# B&R Automation Studio project MotionTestBenchMaster (part 36)

#### FB_MasterAxis.st
```iecst
FUNCTION_BLOCK FB_MasterAxis
	(* The master position is built from the external struct *)
	IF i_xExternalEncoder OR i_xExternalPositionFormat THEN//V4.A.A.1.7.0
		diMasterPosition	:= i_pstExtEncoderPosition;
	ELSE
		diMasterPosition	:= LREAL_TO_DINT(i_pstMasterPositionStruct.VLab_LRealPosition * 100); //0..36000 * 100 to reach 0..3600000
	END_IF

	IF i_uiNumberOfSteps = 0 THEN
		i_uiNumberOfSteps := 1;
	END_IF

	IF i_udiExternalSignalPeriod = 0 THEN
		i_udiExternalSignalPeriod	:= 3600000;
	END_IF

	(* Master communication fault, Master Encoder not referenced *)
	IF eDigitalSynchroStep > SYNCHRO_INIT THEN
		IF NOT i_xEnable THEN	//V4.A.A.1.6.10
			eDigitalSynchroStep := SYNCHRO_INIT;
		ELSIF NOT i_xCmdEnableCurves AND eDigitalSynchroStep < ERROR THEN
			eDigitalSynchroStep	:= ERROR;
		ELSIF fbWriteParID.Error THEN //Read ParID error
			eDigitalSynchroStep	:= ERROR;
		ELSIF fbCyclicWrite_ExtrEncPos.Error	OR fbCyclicWrite_RefExtrEncPos.Error
			OR fbCyclicRead_ScaledPos.Error		OR fbCyclicRead_ModuloPos.Error 		OR fbCyclicRead_RefModuloPos.Error THEN //Cyclic communication error

			eDigitalSynchroStep	:= ERROR;
		END_IF
	END_IF

	fbRTInfo.enable	:= TRUE;	//V4.A.A.1.6.10
	fbRTInfo();	//V4.A.A.1.6.10

	CASE eDigitalSynchroStep OF
		SYNCHRO_INIT:
			i_pstParameter.i_pdiMasterScaledPos	:= ADR(diMasterScaledPos);
			i_pstParameter.i_plrMasterPosition	:= ADR(lrExternalRefPosition);
			i_pstParameter.i_prMasterVelocity	:= ADR(rExternalRefVelocity);
			i_pstParameter.i_xMachineMaster		:= TRUE;

			i_pstParameter.i_uiMasterParId		:= ACP10PAR_CURVE_VALUE_I4 + 1;

			TON_WaitCurveStabilization.PT		:= T#500ms; // Wait for CURVE FBK stable output
			TON_WaitCurveStabilization.IN		:= FALSE;

			fbPeriodicToContinuePosition.i_xEnable 	:= FALSE;

			(* === Parameters for cyclic data exchange between plc and drive === *)
			fbCyclicRead_ScaledPos.Axis				:= i_pAxisADR;
			fbCyclicRead_ScaledPos.ParID			:= ACP10PAR_CURVE_VALUE_I4 +1;
			fbCyclicRead_ScaledPos.DataAddress		:= ADR(diMasterScaledPos);
			fbCyclicRead_ScaledPos.DataType			:= ncPAR_TYP_DINT;
			fbCyclicRead_ScaledPos.Mode				:= mcEVERY_RECORD;
			fbCyclicRead_ScaledPos.Enable			:= FALSE;

			fbCyclicRead_ModuloPos.Axis				:= i_pAxisADR;
			fbCyclicRead_ModuloPos.ParID			:= ACP10PAR_CURVE_VALUE_REL_I4 +1;
			fbCyclicRead_ModuloPos.DataAddress		:= ADR(diMasterModuloPos);
			fbCyclicRead_ModuloPos.DataType			:= ncPAR_TYP_DINT;
			fbCyclicRead_ModuloPos.Mode				:= mcEVERY_RECORD;
			fbCyclicRead_ModuloPos.Enable			:= FALSE;

			fbCyclicWrite_ExtrEncPos.Axis			:= i_pAxisADR;
			fbCyclicWrite_ExtrEncPos.ParID			:= ACP10PAR_VAR_I4_0;
			fbCyclicWrite_ExtrEncPos.DataAddress	:= ADR(diMasterPosToSpt);
			fbCyclicWrite_ExtrEncPos.DataType		:= ncPAR_TYP_DINT;
			fbCyclicWrite_ExtrEncPos.Mode			:= mcEVERY_RECORD;
			fbCyclicWrite_ExtrEncPos.Enable			:= FALSE;

			(* === Non - Filtered parameter computation for positioning error check === *)
			fbCyclicWrite_RefExtrEncPos.Axis		:= i_pAxisADR;
			fbCyclicWrite_RefExtrEncPos.ParID		:= ACP10PAR_VAR_I4_3;
			fbCyclicWrite_RefExtrEncPos.DataAddress	:= ADR(diRefExtrEncPos);
			fbCyclicWrite_RefExtrEncPos.DataType	:= ncPAR_TYP_DINT;
			fbCyclicWrite_RefExtrEncPos.Mode		:= mcEVERY_RECORD;
			fbCyclicWrite_RefExtrEncPos.Enable		:= FALSE;

			fbCyclicRead_RefModuloPos.Axis			:= i_pAxisADR;
			fbCyclicRead_RefModuloPos.ParID			:= ACP10PAR_CURVE_VALUE_REL_I4 +4;
			fbCyclicRead_RefModuloPos.DataAddress	:= ADR(diRefModuloPos);
			fbCyclicRead_RefModuloPos.DataType		:= ncPAR_TYP_DINT;
//			fbCyclicRead_RefModuloPos.Mode			:= mcEVERY_RECORD;	V 1.1
			fbCyclicRead_RefModuloPos.Enable		:= FALSE;

			IF i_xEnable THEN
				eDigitalSynchroStep		:= CURVES_DISABLE;
			END_IF

		CURVES_DISABLE:
			IF NOT fbWriteParID.Busy THEN
				uiCurveMode					:= 0; //DISABLE
				fbWriteParID.Axis			:= i_pAxisADR;
				fbWriteParID.DataAddress	:= ADR(uiCurveMode);
				fbWriteParID.DataType		:= ncPAR_TYP_UINT;
				fbWriteParID.ParID			:= ACP10PAR_CURVE_MODE + 0;
				fbWriteParID.Execute		:= TRUE;
			END_IF

			IF fbWriteParID.Done AND fbWriteParID.ParID = ACP10PAR_CURVE_MODE + 0 THEN
				fbWriteParID.Execute	:= FALSE;
				eDigitalSynchroStep		:= CURVES_DISABLE_1;
			END_IF

		CURVES_DISABLE_1:
			IF NOT fbWriteParID.Busy THEN
				uiCurveMode					:= 0; //DISABLE
				fbWriteParID.DataAddress	:= ADR(uiCurveMode);
				fbWriteParID.DataType		:= ncPAR_TYP_UINT;
				fbWriteParID.ParID			:= ACP10PAR_CURVE_MODE + 1;
				fbWriteParID.Execute		:= TRUE;
			END_IF

			IF fbWriteParID.Done AND fbWriteParID.ParID = ACP10PAR_CURVE_MODE + 1 THEN
				fbWriteParID.Execute	:= FALSE;
				eDigitalSynchroStep		:= CURVES_DISABLE_2;
			END_IF

		CURVES_DISABLE_2:
			IF NOT fbWriteParID.Busy THEN
				uiCurveMode					:= 0; //DISABLE
				fbWriteParID.DataAddress	:= ADR(uiCurveMode);
				fbWriteParID.DataType		:= ncPAR_TYP_UINT;
				fbWriteParID.ParID			:= ACP10PAR_CURVE_MODE + 3;
				fbWriteParID.Execute		:= TRUE;
			END_IF

			IF fbWriteParID.Done AND fbWriteParID.ParID = ACP10PAR_CURVE_MODE + 3 THEN
				fbWriteParID.Execute	:= FALSE;
				eDigitalSynchroStep		:= CURVES_DISABLE_3;
			END_IF

		CURVES_DISABLE_3:
			IF NOT fbWriteParID.Busy THEN
				uiCurveMode					:= 0; //DISABLE
				fbWriteParID.DataAddress	:= ADR(uiCurveMode);
				fbWriteParID.DataType		:= ncPAR_TYP_UINT;
				fbWriteParID.ParID			:= ACP10PAR_CURVE_MODE + 4;
				fbWriteParID.Execute		:= TRUE;
			END_IF

			IF fbWriteParID.Done AND fbWriteParID.ParID = ACP10PAR_CURVE_MODE + 4 THEN
				TON_WaitCurveStabilization.IN	:= FALSE;
				fbWriteParID.Execute			:= FALSE;
				eDigitalSynchroStep				:= ZERO_OFFSET;
			END_IF

		(* In order to be sure that the OFFSET is zero at the startup the value is force *)
		ZERO_OFFSET:
			IF NOT fbWriteParID.Busy THEN
				q_diOffsetModuloPos			:= 0;
				fbWriteParID.DataAddress	:= ADR(q_diOffsetModuloPos);
				fbWriteParID.DataType		:= ncPAR_TYP_DINT;
				fbWriteParID.ParID			:= ACP10PAR_VAR_I4_1 +0;
				fbWriteParID.Execute		:= TRUE;
			END_IF

			IF fbWriteParID.Done AND fbWriteParID.ParID = ACP10PAR_VAR_I4_1 + 0 THEN
				fbWriteParID.Execute 	:= FALSE;
				q_xPositionRestored 	:= TRUE;
				eDigitalSynchroStep 	:= WRITE_MA_PERIOD;
			END_IF

		WRITE_MA_PERIOD:
			IF NOT fbWriteParID.Busy THEN
				diMasterPeriod				:= i_udiExternalSignalPeriod;
				fbWriteParID.Axis			:= i_pAxisADR;
				fbWriteParID.DataAddress	:= ADR(diMasterPeriod);
				fbWriteParID.DataType		:= ncPAR_TYP_DINT;
				fbWriteParID.ParID			:= ACP10PAR_CURVE_X_FACTOR + 0;
				fbWriteParID.Execute		:= TRUE;
			END_IF

			IF fbWriteParID.Done AND fbWriteParID.ParID = ACP10PAR_CURVE_X_FACTOR + 0 THEN
				fbWriteParID.Execute	:= FALSE;
				eDigitalSynchroStep		:= WRITE_MA_PERIOD_1;
			END_IF

		WRITE_MA_PERIOD_1:
			IF NOT fbWriteParID.Busy THEN
				diMasterPeriod				:= i_udiExternalSignalPeriod;
				fbWriteParID.Axis			:= i_pAxisADR;
				fbWriteParID.DataAddress	:= ADR(diMasterPeriod);
				fbWriteParID.DataType		:= ncPAR_TYP_DINT;
				fbWriteParID.ParID			:= ACP10PAR_CURVE_X_FACTOR + 3;
				fbWriteParID.Execute		:= TRUE;
			END_IF

			IF fbWriteParID.Done AND fbWriteParID.ParID = ACP10PAR_CURVE_X_FACTOR + 3 THEN
				fbWriteParID.Execute	:= FALSE;
				eDigitalSynchroStep		:= WRITE_SL_PERIOD;
			END_IF

		WRITE_SL_PERIOD:
			IF NOT fbWriteParID.Busy THEN
				diSlavePeriod				:= i_uiNumberOfSteps * 360 * c_uiAxisFactor;
				fbWriteParID.Axis			:= i_pAxisADR;
				fbWriteParID.DataAddress	:= ADR(diSlavePeriod);
				fbWriteParID.DataType		:= ncPAR_TYP_DINT;
				fbWriteParID.ParID			:= ACP10PAR_CURVE_Y_FACTOR + 0;
				fbWriteParID.Execute		:= TRUE;
			END_IF

			IF fbWriteParID.Done AND fbWriteParID.ParID = ACP10PAR_CURVE_Y_FACTOR + 0 THEN
				fbWriteParID.Execute	:= FALSE;
				eDigitalSynchroStep		:= WRITE_SL_PERIOD_1;
			END_IF

		WRITE_SL_PERIOD_1:
			IF NOT fbWriteParID.Busy THEN
				diSlavePeriod				:= i_uiNumberOfSteps * 360 * c_uiAxisFactor;
				fbWriteParID.Axis			:= i_pAxisADR;
				fbWriteParID.DataAddress	:= ADR(diSlavePeriod);
				fbWriteParID.DataType		:= ncPAR_TYP_DINT;
				fbWriteParID.ParID			:= ACP10PAR_CURVE_Y_FACTOR + 3;
				fbWriteParID.Execute		:= TRUE;
			END_IF

			IF fbWriteParID.Done AND fbWriteParID.ParID = ACP10PAR_CURVE_Y_FACTOR + 3 THEN
				fbWriteParID.Execute	:= FALSE;
				eDigitalSynchroStep		:= INIT_FILTERS;
			END_IF

		INIT_FILTERS:
			lrFilterTime 	:= UINT_TO_LREAL(i_uiFilteringCoefficient) * c_rTf_min; (* s *)
			lrExtrTime 		:= (UDINT_TO_LREAL(fbRTInfo.cycle_time) / 1E6) * UINT_TO_LREAL(i_uiNumberOfEplCycles) + c_timCompensationIPL; (* s *)	//V4.A.A.1.6.10

			(* Periodic to continue position enable *)
			fbPeriodicToContinuePosition.i_xEnable 	:= TRUE;

			(* Reference filter enable *)
			(* The enable is done only in case of i_uiFilteringCoefficient > 0 *)

			fbEXTR_RefFilter.Enable		:= lrFilterTime > 0;

			(* Extrapolation filter enable *)
			fbPT1_EncFilter.Enable 		:= fbEXTR_RefFilter.Enable;

			IF i_udiExternalSignalPeriod > 0 THEN
				diInitialOffset	:= diMasterPosition - (diMasterPosition MOD UDINT_TO_DINT(i_udiExternalSignalPeriod));
			END_IF

			IF fbEXTR_RefFilter.Enable AND fbPT1_EncFilter.Enable THEN
				IF fbPT1_EncFilter.Valid THEN
					fbEXTR_EncFilter.Enable	:= TRUE;
					IF fbEXTR_EncFilter.Valid AND fbEXTR_RefFilter.Valid THEN
						TON_WaitCurveStabilization.IN	:= FALSE;
						eDigitalSynchroStep 			:= DISABLE_IPL;
					END_IF
				END_IF
			ELSE
				TON_WaitCurveStabilization.IN	:= FALSE;
				eDigitalSynchroStep 			:= DISABLE_IPL;
			END_IF

		DISABLE_IPL:
			IF NOT fbWriteParID.Busy THEN
				uiIPLMode					:= 0;
				fbWriteParID.Axis			:= i_pAxisADR;
				fbWriteParID.DataAddress	:= ADR(uiIPLMode);
				fbWriteParID.DataType		:= ncPAR_TYP_UINT;
				fbWriteParID.ParID			:= ACP10PAR_IPL_MODE + 0;
				fbWriteParID.Execute		:= TRUE;
			END_IF

			TON_WaitCurveStabilization.IN	:= fbWriteParID.Done;
			TON_WaitCurveStabilization.PT	:= T#0.5S;

			IF TON_WaitCurveStabilization.Q AND fbWriteParID.ParID = ACP10PAR_IPL_MODE + 0 THEN
				fbWriteParID.Execute	:= FALSE;
				eDigitalSynchroStep		:= INIT_CYCLIC_READ_WRITE;
			END_IF

		INIT_CYCLIC_READ_WRITE:
			fbCyclicWrite_ExtrEncPos.Enable		:= TRUE;
			fbCyclicWrite_RefExtrEncPos.Enable	:= TRUE;

			fbCyclicRead_ScaledPos.Enable		:= TRUE;
			fbCyclicRead_ModuloPos.Enable 		:= TRUE;
			fbCyclicRead_RefModuloPos.Enable	:= TRUE;

			q_xCyclicComValid	:= fbCyclicWrite_ExtrEncPos.Valid AND fbCyclicWrite_RefExtrEncPos.Valid AND fbCyclicRead_ScaledPos.Valid AND
									fbCyclicRead_ModuloPos.Valid AND fbCyclicRead_RefModuloPos.Valid;

			IF fbCyclicWrite_ExtrEncPos.Error OR fbCyclicWrite_RefExtrEncPos.Error OR fbCyclicRead_ScaledPos.Error OR fbCyclicRead_ModuloPos.Error OR fbCyclicRead_RefModuloPos.Error THEN
				q_xCyclicComValid 	:= FALSE;
				eDigitalSynchroStep := ERROR;
			ELSIF q_xCyclicComValid THEN
				TON_WaitCurveStabilization.IN	:= FALSE;
				eDigitalSynchroStep 			:= WRITE_IPL_CYCLIE_TIME;
			END_IF

		WRITE_IPL_CYCLIE_TIME:
			IF NOT fbWriteParID.Busy THEN

				IF i_xExternalEncoder THEN
					udiCycleTime				:= fbRTInfo.cycle_time * 10;	//V4.A.A.1.6.10
				ELSIF i_xExternalPositionFormat THEN//V4.A.A.1.7.0
					udiCycleTime				:= fbRTInfo.cycle_time * 2;//V4.A.A.1.7.0
				ELSE
					udiCycleTime				:= fbRTInfo.cycle_time;	//V4.A.A.1.6.10
				END_IF

				fbWriteParID.Axis			:= i_pAxisADR;
				fbWriteParID.DataAddress	:= ADR(udiCycleTime);
				fbWriteParID.DataType		:= ncPAR_TYP_UDINT;
				fbWriteParID.ParID			:= ACP10PAR_IPL_CYCLE_TIME + 0;
				fbWriteParID.Execute		:= TRUE;
			END_IF

			IF fbWriteParID.Done AND fbWriteParID.ParID = ACP10PAR_IPL_CYCLE_TIME + 0 THEN
				fbWriteParID.Execute	:= FALSE;
				eDigitalSynchroStep		:= ENABLE_IPL;
			END_IF

		ENABLE_IPL:
			IF NOT fbWriteParID.Busy THEN
				uiIPLMode					:= 1;
				fbWriteParID.Axis			:= i_pAxisADR;
				fbWriteParID.DataAddress	:= ADR(uiIPLMode);
				fbWriteParID.DataType		:= ncPAR_TYP_UINT;
				fbWriteParID.ParID			:= ACP10PAR_IPL_MODE + 0;
				fbWriteParID.Execute		:= TRUE;
			END_IF

			TON_WaitCurveStabilization.IN	:= fbWriteParID.Done;
			TON_WaitCurveStabilization.PT	:= T#0.5S;

			IF TON_WaitCurveStabilization.Q AND fbWriteParID.ParID = ACP10PAR_IPL_MODE + 0 THEN
				fbWriteParID.Execute	:= FALSE;
				eDigitalSynchroStep		:= CURVES_ENABLE;
			END_IF

		CURVES_ENABLE:
			IF NOT fbWriteParID.Busy THEN
				uiCurveMode					:= 2;
				fbWriteParID.Axis			:= i_pAxisADR;
				fbWriteParID.DataAddress	:= ADR(uiCurveMode);
				fbWriteParID.DataType		:= ncPAR_TYP_UINT;
				fbWriteParID.ParID			:= ACP10PAR_CURVE_MODE + 0;
				fbWriteParID.Execute		:= TRUE;
			END_IF

			IF fbWriteParID.Done AND fbWriteParID.ParID = ACP10PAR_CURVE_MODE + 0 THEN
				fbWriteParID.Execute	:= FALSE;
				eDigitalSynchroStep		:= CURVES_ENABLE_1;
			END_IF

		CURVES_ENABLE_1:
			IF NOT fbWriteParID.Busy THEN
				uiCurveMode					:= 2;
				fbWriteParID.DataAddress	:= ADR(uiCurveMode);
				fbWriteParID.DataType		:= ncPAR_TYP_UINT;
				fbWriteParID.ParID			:= ACP10PAR_CURVE_MODE + 1;
				fbWriteParID.Execute		:= TRUE;
			END_IF

			IF fbWriteParID.Done AND fbWriteParID.ParID = ACP10PAR_CURVE_MODE + 1 THEN
				fbWriteParID.Execute	:= FALSE;
				eDigitalSynchroStep		:= CURVES_ENABLE_2;
			END_IF

		CURVES_ENABLE_2:
			IF NOT fbWriteParID.Busy THEN
				uiCurveMode					:= 2;
				fbWriteParID.DataAddress	:= ADR(uiCurveMode);
				fbWriteParID.DataType		:= ncPAR_TYP_UINT;
				fbWriteParID.ParID			:= ACP10PAR_CURVE_MODE + 3;
				fbWriteParID.Execute		:= TRUE;
			END_IF

			IF fbWriteParID.Done AND fbWriteParID.ParID = ACP10PAR_CURVE_MODE + 3 THEN
				fbWriteParID.Execute	:= FALSE;
				eDigitalSynchroStep		:= CURVES_ENABLE_3;
			END_IF

		CURVES_ENABLE_3:
			IF NOT fbWriteParID.Busy THEN
				uiCurveMode					:= 2;
				fbWriteParID.DataAddress	:= ADR(uiCurveMode);
				fbWriteParID.DataType		:= ncPAR_TYP_UINT;
				fbWriteParID.ParID			:= ACP10PAR_CURVE_MODE + 4;
				fbWriteParID.Execute		:= TRUE;
			END_IF

			IF fbWriteParID.Done AND fbWriteParID.ParID = ACP10PAR_CURVE_MODE + 4 THEN
				fbWriteParID.Execute			:= FALSE;
				TON_WaitCurveStabilization.IN	:= FALSE;
				eDigitalSynchroStep				:= WAIT_CURVES_STABILIZATION;
			END_IF

		WAIT_CURVES_STABILIZATION:
			IF diOldScaledPos = diMasterScaledPos AND diOldModuloPos = diMasterModuloPos THEN
				TON_WaitCurveStabilization.IN	:= TRUE;
				IF TON_WaitCurveStabilization.Q THEN
					TON_WaitCurveStabilization.IN	:= FALSE;
					q_xPositionValid 				:= TRUE;
					eDigitalSynchroStep				:= RESTORE_CALIBRATION_OFFSET;
				END_IF
			ELSE
				TON_WaitCurveStabilization.IN := FALSE;
				diOldScaledPos := diMasterScaledPos;
				diOldModuloPos := diMasterModuloPos;
			END_IF

		RESTORE_CALIBRATION_OFFSET:
			IF NOT fbWriteParID.Busy THEN
				q_diOffsetModuloPos			:= i_pstAbsEncPerm.diAbsEncOffset;
				fbWriteParID.DataAddress	:= ADR(q_diOffsetModuloPos);
				fbWriteParID.DataType		:= ncPAR_TYP_DINT;
				fbWriteParID.ParID			:= ACP10PAR_VAR_I4_1 +0;
				fbWriteParID.Execute		:= TRUE;
			END_IF

			IF fbWriteParID.Done AND fbWriteParID.ParID = ACP10PAR_VAR_I4_1 + 0 THEN
				fbWriteParID.Execute := FALSE;

				q_xPositionRestored := TRUE;
				eDigitalSynchroStep := ABS_ENC_READY;
			END_IF

		ABS_ENC_READY:
			q_xCyclicComValid	:= fbCyclicWrite_ExtrEncPos.Valid AND fbCyclicWrite_RefExtrEncPos.Valid AND fbCyclicRead_ScaledPos.Valid AND
									fbCyclicRead_ModuloPos.Valid AND fbCyclicRead_RefModuloPos.Valid;

			IF NOT q_xCyclicComValid OR NOT i_xCmdEnableCurves THEN
				eDigitalSynchroStep		:= ERROR;
			ELSIF i_pstStatus.q_stMainAxisStatus.q_xSynchroWithOffset AND i_pstCmd.i_xPhaseCompensation THEN //V4.A.A.1.6.10
				eDigitalSynchroStep		:= OFFSET_RESET;
			ELSIF i_xCmdHoming THEN
				eDigitalSynchroStep		:= CALIBRATION;
			END_IF

		OFFSET_RESET:
			q_diOffsetModuloPos	:= REAL_TO_DINT(i_pstAxisHome.rPhaseOffsetValue * c_uiAxisFactor) + i_pstAbsEncPerm.diAbsEncOffset;

			i_pstAxisHome.rPhaseOffsetValue		:= 0;
			i_pstAbsEncPerm.diAbsEncOffset		:= q_diOffsetModuloPos;
			i_pstAbsEncPerm.xCalibrationDone	:= FALSE;
			eDigitalSynchroStep					:= WRITE_NEW_CALIBRATION_VALUE;

		CALIBRATION:
			q_diOffsetModuloPos := LREAL_TO_DINT(i_pstStatus.q_stMainAxisStatus.q_lrPosition * c_uiAxisFactor) - diRefModuloPos;

			IF q_diOffsetModuloPos < 0 THEN
				q_diOffsetModuloPos := q_diOffsetModuloPos + 36000;
			END_IF

			i_pstAbsEncPerm.diAbsEncOffset		:= q_diOffsetModuloPos;
			i_pstAbsEncPerm.xCalibrationDone	:= FALSE;

			eDigitalSynchroStep 	:= WRITE_NEW_CALIBRATION_VALUE;

		WRITE_NEW_CALIBRATION_VALUE:
			IF NOT fbWriteParID.Busy THEN
				fbWriteParID.Axis			:= i_pAxisADR;
				fbWriteParID.DataAddress	:= ADR(q_diOffsetModuloPos);
				fbWriteParID.DataType		:= ncPAR_TYP_DINT;
				fbWriteParID.ParID			:= ACP10PAR_VAR_I4_1;
				fbWriteParID.Execute		:= TRUE;
			END_IF

			IF fbWriteParID.Done AND fbWriteParID.ParID = ACP10PAR_VAR_I4_1 AND NOT i_pstCmd.i_xPhaseCompensation AND NOT i_xCmdHoming THEN
				fbWriteParID.Execute 				:= FALSE;
				i_pstAbsEncPerm.xCalibrationDone	:= TRUE;
				q_xPositionRestored					:= TRUE;
				eDigitalSynchroStep					:= WAIT_CURVES_STABILIZATION;
			END_IF

		(*****************************************)
		ERROR:
			q_xPositionRestored						:= FALSE;
			q_xCyclicComValid						:= FALSE;
			q_xPositionValid  						:= FALSE;

			TON_WaitCurveStabilization.IN 			:= FALSE;
			fbPeriodicToContinuePosition.i_xEnable 	:= FALSE;

			IF i_pstCmd.i_xErrorReset THEN
				fbCyclicWrite_ExtrEncPos.Enable		:= FALSE;
				fbCyclicWrite_RefExtrEncPos.Enable	:= FALSE;

				fbCyclicRead_ScaledPos.Enable		:= FALSE;
				fbCyclicRead_ModuloPos.Enable 		:= FALSE;
				fbCyclicRead_RefModuloPos.Enable	:= FALSE;

				fbPT1_EncFilter.Enable 	:= FALSE;
				fbEXTR_EncFilter.Enable	:= FALSE;
				fbEXTR_RefFilter.Enable	:= FALSE;
				IF fbWriteParID.Error THEN
					fbWriteParID.Execute := FALSE;
				END_IF
			END_IF

			IF NOT fbCyclicWrite_ExtrEncPos.Error AND NOT fbCyclicWrite_RefExtrEncPos.Error AND NOT fbCyclicRead_ScaledPos.Error AND
				NOT fbCyclicRead_ModuloPos.Error AND NOT fbCyclicRead_RefModuloPos.Error AND NOT fbWriteParID.Error THEN

				eDigitalSynchroStep := ERROR_1;
			END_IF

		ERROR_1: (* Wait Master data are OK *)
			IF i_xCmdEnableCurves THEN
				eDigitalSynchroStep := CURVES_DISABLE;
			END_IF
	END_CASE

	(* Timer for curve stabilization *)
	TON_WaitCurveStabilization();

	fbWriteParID();

	fbCyclicRead_ScaledPos();
	fbCyclicRead_ModuloPos();
	fbCyclicRead_RefModuloPos();
	fbCyclicWrite_ExtrEncPos();
	fbCyclicWrite_RefExtrEncPos();

	(* Periodic TO Continue DINT position *)
	IF NOT i_xExternalEncoder THEN
		fbPeriodicToContinuePosition.i_diInPosition	:= diMasterPosition;
		fbPeriodicToContinuePosition.i_udiPeriod	:= i_udiExternalSignalPeriod;
		fbPeriodicToContinuePosition();
	END_IF

	IF fbPT1_EncFilter.Enable THEN
		IF NOT i_xExternalEncoder THEN (* External Value filtering *)
			fbPT1_EncFilter.T1	:= lrFilterTime;
			fbPT1_EncFilter.U	:= fbPeriodicToContinuePosition.q_diPosition;
		ELSE (* External Value filtering *)
			fbPT1_EncFilter.T1	:= lrFilterTime;
			fbPT1_EncFilter.U	:= (diMasterPosition - diInitialOffset);
		END_IF

		fbPT1_EncFilter();

		(* External value extrapolation *)
		fbEXTR_EncFilter.T_ext	:= lrExtrTime + lrFilterTime;
		fbEXTR_EncFilter.U		:= fbPT1_EncFilter.X;
		fbEXTR_EncFilter();

		(* External Value filtering *)
		IF NOT i_xExternalEncoder THEN
			diMasterPosToSpt	 	:= fbEXTR_EncFilter.X;
		ELSE
			uiMasterPositionSampling := uiMasterPositionSampling + 1;	//v1.2
			IF uiMasterPositionSampling >= 10 THEN				//v1.2
				diMasterPosToSpt	 	:= fbEXTR_EncFilter.X;
				uiMasterPositionSampling	:= 0;			//v1.2
			END_IF
		END_IF

		(* Non-filtered position extrapolation *)
		IF NOT i_xExternalEncoder THEN (* External Value filtering *)
			fbEXTR_RefFilter.T_ext	:= lrExtrTime;
			fbEXTR_RefFilter.U	:= fbPeriodicToContinuePosition.q_diPosition;
		ELSE (* External Value filtering *)
			fbEXTR_RefFilter.T_ext	:= lrExtrTime;
			fbEXTR_RefFilter.U	:= (diMasterPosition - diInitialOffset);
		END_IF
		fbEXTR_RefFilter();

		diRefExtrEncPos			:= fbEXTR_RefFilter.X;

		(* Extrapolation error computing *)
		IF EDGEPOS(q_xPositionValid) THEN
			diRefModuloOffset := diMasterModuloPos - diRefModuloPos;
		END_IF

		q_diRefPosError := diMasterModuloPos - diRefModuloPos - diRefModuloOffset;

		IF ABS(q_diRefPosError + 360 * c_uiAxisFactor) < ABS(q_diRefPosError) THEN
			q_diRefPosError := q_diRefPosError + 360 * c_uiAxisFactor;
		ELSIF ABS(q_diRefPosError - 360 * c_uiAxisFactor) < ABS(q_diRefPosError) THEN
			q_diRefPosError := q_diRefPosError - 360 * c_uiAxisFactor;
		END_IF
	ELSIF NOT i_xExternalEncoder THEN
		diMasterPosToSpt	:= fbPeriodicToContinuePosition.q_diPosition;
		diRefExtrEncPos		:= fbPeriodicToContinuePosition.q_diPosition;
	ELSE
		uiMasterPositionSampling := uiMasterPositionSampling + 1;	//v1.2
		IF uiMasterPositionSampling >= 10 THEN				//v1.2
			diMasterPosToSpt	 	:= diMasterPosition;
			uiMasterPositionSampling	:= 0;			//v1.2
		END_IF

		diRefExtrEncPos		:= diMasterPosition;
	END_IF

	(* External reference position and velocity *)
	lrExternalRefPosition  := UDINT_TO_LREAL(diMasterModuloPos) / c_uiAxisFactor;

	fbVelocity.i_diPosition	:= diMasterScaledPos;
	fbVelocity();
	rExternalRefVelocity	:= fbVelocity.q_rVelocity / c_uiAxisFactor;
END_FUNCTION_BLOCK
```

#### FB_Step2PeriodicPosition.st
```iecst
(* From a step signal a periodic signal is created *)
FUNCTION_BLOCK FB_PeriodicPosition
	IF NOT i_xEnable OR i_rPeriod <=0 THEN
		usiStep				:= 0;
		q_xPositionValid	:= FALSE;
	ELSE
		CASE usiStep OF
			0:
				q_xPositionValid	:= FALSE;
				q_rPeriodicPosition	:= 0;
				rPosition			:= 0;

				IF i_xEnable THEN
					usiStep	:= 10;
				END_IF

			10:
				IF EDGEPOS(i_xResetPostion) THEN
					q_xPositionValid	:= TRUE;
					rPosition			:= i_rAxisPosition;
					q_rPeriodicPosition	:= i_rAxisPosition;
					usiStep				:= 20;
				END_IF

			20:
				rDeltaPos	:= i_rAxisPosition - rPosition;
				// If the difference between the old axis and the current axis position
				// If greater than 180° it means that we overlapped the period
				IF ABS(rDeltaPos) > 180 THEN
					IF rDeltaPos > 0 THEN
						rDeltaPos	:= rDeltaPos - 360;
					ELSE
						rDeltaPos	:= rDeltaPos + 360;
					END_IF
				END_IF

				q_rPeriodicPosition	:= FC_RealReminder(q_rPeriodicPosition + rDeltaPos, i_rPeriod, 0);
				rPosition			:= i_rAxisPosition;

				IF i_xResetPostion	THEN
					usiStep	:= 0;
				END_IF
		END_CASE
	END_IF
END_FUNCTION_BLOCK
```

#### FB_CamGenerator.st
```iecst
(* Cam Generator Function Block *)
FUNCTION_BLOCK FB_CamGenerator
	IF i_xEnable AND i_usiNumberOfPulse > 0 THEN
		IF i_usiNumberOfPulse = 1 AND i_rOnPosition <> i_rOffPosition THEN
			rAdvPosition		:= i_rAdvanceTime * i_prAxisVelocity / 1000.0;
			q_xAdvError			:= (ABS(rAdvPosition) >= 360);

			i_pxPointerStepAdv	:= ((i_rOnPosition - rAdvPosition) < 0);

			rOnPositionA		:= FC_RealReminder(i_rOnPosition - rAdvPosition,	360.0, 0);
			rOffPositionA		:= FC_RealReminder(i_rOffPosition - rAdvPosition,	360.0, 0);

			(* CAM A GENERATION *)
			IF(rOnPositionA < rOffPositionA) THEN
				xCamValueA	:= (i_plrAxisPosition >= rOnPositionA) AND (i_plrAxisPosition < rOffPositionA);
			ELSE
				xCamValueA	:= i_plrAxisPosition >= rOnPositionA OR i_plrAxisPosition < rOffPositionA;
			END_IF

			IF xCamValueA <> xOldCamValueA THEN
				rTempReal	:= SEL(xCamValueA, rOffPositionA, rOnPositionA);
				rTempReal	:= rTempReal - LREAL_TO_REAL(i_plrAxisPosition);
				IF ABS(rTempReal) > 0.5 AND ABS(rTempReal) < 359.5 THEN
					xOldCamValueA := xCamValueA;
				END_IF
			END_IF

			(* CAM B GENERATION *)
			IF i_rOnPositionB <> 0 AND i_rOffPositionB <> 0 THEN
				rOnPositionB		:= FC_RealReminder(i_rOnPositionB - rAdvPosition,	360.0, 0);
				rOffPositionB		:= FC_RealReminder(i_rOffPositionB - rAdvPosition,	360.0, 0);
				IF(rOnPositionB < rOffPositionB) THEN
					xCamValueB	:= (i_plrAxisPosition >= rOnPositionB) AND (i_plrAxisPosition < rOffPositionB);
				ELSE
					xCamValueB	:= i_plrAxisPosition >= rOnPositionB OR i_plrAxisPosition < rOffPositionB;
				END_IF

				IF xCamValueB <> xOldCamValueB THEN
					rTempReal	:= SEL(xCamValueB, rOffPositionB, rOnPositionB);
					rTempReal	:= rTempReal - LREAL_TO_REAL(i_plrAxisPosition);
					IF ABS(rTempReal) > 0.5 AND ABS(rTempReal) < 359.5 THEN
						xOldCamValueB	:=	xCamValueB;
					END_IF
				END_IF

				(* Debounce *)
				CASE usiStep OF
					0:(* INIT *)
						usiStep := 100;

					100:(* WAIT FOR CAM A RAISING EDGE *)
						IF xCamValueA THEN
							i_pxPointerOutput := TRUE;
							usiStep := 110;
						END_IF

					110:(* WAIT FOR CAM B FALLING EDGE *)
						IF NOT xCamValueB THEN
							usiStep := 120;
						END_IF

					120:(*  WAIT FOR CAM A FALLING EDGE *)
						IF NOT xCamValueA THEN
							i_pxPointerOutput := FALSE;
							usiStep := 130;
						END_IF

					130:(* WAIT FOR CAM B RAISING EDGE *)
						IF xCamValueB THEN
							usiStep := 100;
						END_IF

					ELSE
						usiStep := 200;
				END_CASE
			ELSE
				(* Simple cam A generator *)
				i_pxPointerOutput	:= xOldCamValueA;
			END_IF
		ELSIF i_usiNumberOfPulse <= 10 THEN
			i_pxPointerStepAdv	:= FALSE;
			i_pxPointerOutput	:= FC_RealReminder(LREAL_TO_REAL(i_plrAxisPosition), 360.0 / i_usiNumberOfPulse, 0) >= 180.0 / i_usiNumberOfPulse;
		END_IF
	ELSE
		i_pxPointerOutput	:= FALSE;
		q_xAdvError			:= FALSE;
	END_IF
END_FUNCTION_BLOCK

(* Cam Generator Function Block *)
FUNCTION_BLOCK FB_CamGenerator_v2
	IF i_xEnable AND i_usiNumberOfPulse > 0 THEN
		IF i_usiNumberOfPulse = 1 AND i_rOnPosition <> i_rOffPosition THEN
			rPosition			:= DINT_TO_REAL(i_pdiAxisPosition MOD 36000) / 100.0;
			rAdvPosition		:= i_rAdvanceTime * i_prAxisVelocity / 100000.0; //v1.4
			q_xAdvError			:= (ABS(rAdvPosition) >= 360);

			i_pxPointerStepAdv	:= ((i_rOnPosition - rAdvPosition) < 0);

			rOnPosition		:= FC_RealReminder(i_rOnPosition - rAdvPosition,	360.0, 0);
			rOffPosition	:= FC_RealReminder(i_rOffPosition - rAdvPosition,	360.0, 0);

			(* CAM GENERATION *)
			IF(rOnPosition < rOffPosition) THEN
				xCamValue	:= (rPosition >= rOnPosition) AND (rPosition < rOffPosition);
			ELSE
				xCamValue	:= rPosition >= rOnPosition OR rPosition < rOffPosition;
			END_IF

			IF xCamValue <> xOldCamValue THEN
				rTempReal	:= SEL(xCamValue, rOffPosition, rOnPosition);
				rTempReal	:= rTempReal - rPosition;
				IF ABS(rTempReal) > 0.5 AND ABS(rTempReal) < 359.5 THEN
					xOldCamValue := xCamValue;
				END_IF
			END_IF

			i_pxPointerOutput	:= xOldCamValue;
		ELSIF i_usiNumberOfPulse <= 10 THEN
			i_pxPointerStepAdv	:= FALSE;
			rPosition			:= DINT_TO_REAL(i_pdiAxisPosition MOD 36000) / 100.0;
			i_pxPointerOutput	:= FC_RealReminder(rPosition, 360.0 / i_usiNumberOfPulse, 0) >= 180.0 / i_usiNumberOfPulse;
		END_IF
	ELSE
		i_pxPointerOutput	:= FALSE;
		q_xAdvError			:= FALSE;
	END_IF
END_FUNCTION_BLOCK
```

#### FB_ExceptionAlarmX.st
```iecst
(* Fb for mananging alarms *)
FUNCTION_BLOCK FB_ExceptionAlarmX
	IF i_pxInitCoreDone THEN
		IF i_xConditions AND NOT xAlarmActive THEN
			xAlarmActive := TRUE;
			MpAlarmXSet(MpLink := i_pstMpAlarmXLink, Name := i_psAlarmName);
		ELSIF NOT i_xConditions AND xAlarmActive THEN
			IF i_pxAcknowledge OR i_xAutoAck THEN
				xAlarmActive := FALSE;
				MpAlarmXReset(MpLink := i_pstMpAlarmXLink, Name := i_psAlarmName);
			END_IF
		END_IF
		q_xAlarmActive := xAlarmActive;
	END_IF
END_FUNCTION_BLOCK
```

#### FB_Position2Velocity.st
```iecst
FUNCTION_BLOCK FB_Position2Velocity
	fbRTInfo(enable := TRUE);
	adiBuffer[uiCount]	:= i_diPosition;
	IF uiCount > 0 THEN
		arBufferVel[uiCount] := DINT_TO_REAL((i_diPosition - adiBuffer[uiCount - 1])) / (DINT_TO_REAL(fbRTInfo.cycle_time) * 1E-6);
	ELSE
		arBufferVel[uiCount] := DINT_TO_REAL((i_diPosition - adiBuffer[c_usiNSample - 1])) / (DINT_TO_REAL(fbRTInfo.cycle_time) * 1E-6);
	END_IF

	uiCount 	:= (uiCount + 1) MOD c_usiNSample;
	rInternal	:= 0;

	FOR i := 0 TO c_usiNSample - 1 DO
		rInternal	:= rInternal + arBufferVel[i];
	END_FOR

	q_rVelocity := rInternal / c_usiNSample;
END_FUNCTION_BLOCK
```

#### FB_Periodic2ContinuePosition.st
```iecst
FUNCTION_BLOCK FB_Periodic2ContinuePosition
	IF NOT i_xEnable THEN
		xActive 		:= FALSE;
		diOldInPosition := 0;
		q_diPosition	:= 0;
		RETURN;
	ELSIF NOT xActive THEN
		xActive 		:= TRUE;
		q_diPosition	:= i_diInPosition;
		diOldInPosition := i_diInPosition;
	ELSE
		(* Continue DINT position calculation *)
		IF ABS(i_diInPosition - diOldInPosition) < UDINT_TO_DINT(i_udiPeriod / 2) THEN
			q_diPosition		:= q_diPosition + (i_diInPosition - diOldInPosition);
		ELSIF i_diInPosition < diOldInPosition THEN
			q_diPosition		:= q_diPosition + i_udiPeriod + (i_diInPosition - diOldInPosition);
		ELSE
			q_diPosition		:= q_diPosition - i_udiPeriod + (i_diInPosition - diOldInPosition);
		END_IF
		diOldInPosition 	:= i_diInPosition;
	END_IF
END_FUNCTION_BLOCK
```

#### FB_EncEmul.st
```iecst
(*********************************************************************************
 * Copyright:
 * Author:    		EncoderEmulationManagement
 * Created:  		July 4, 2016/2:37 PM
 * HELP REFERENCE:  ncsoftware/acp10_drivefunctions/acp10_drivefunctions-63-15.html
 *********************************************************************************)

(* Encoder Emulation on 8BAC130.001-1 plug-in module*)
FUNCTION_BLOCK FB_EncEmul
	IF i_pstEncEmulAxis.nc_obj_inf.node_nr > 0 AND i_pstEncEmulAxis.network.phase  <> 90 AND uiStep > 0 THEN
		uiStep := 950;
	ELSIF fbAxisError.Error	THEN
		uiStep := 960;
	ELSIF fbAxisError.Enable AND (fbAxisError.FunctionBlockErrorCount > 0 OR fbAxisError.AxisErrorCount > 0 ) THEN
		uiStep := 970;
	END_IF

	CASE uiStep OF
		0:(* DISABLE *)
			q_xError 					:= FALSE;
			q_xActive					:= FALSE;
			fbReadParID.Execute 		:= FALSE;
			fbWriteParID_Text.Execute 	:= FALSE;
			fbWriteParID.Execute 		:= FALSE;

			IF NOT i_xErrorReset AND i_pstEncEmulAxis.network.phase  = 90 AND i_pstEncEmulAxis.nc_obj_inf.node_nr > 0 THEN
				fbAxisError.Axis	:= ADR(i_pstEncEmulAxis);
				fbAxisError.Mode	:= mcNO_TEXT + mcACKNOWLEDGE_ALL;
				fbAxisError.Enable	:= TRUE; //V4.A.A.1.6.13
				uiStep				:= 10;
			END_IF

		(**************************** CONFIGURE ENCODER EMULATION ****************************)
		10:(* ENCODER TYPE CONFIG *)
			IF NOT fbWriteParID.Execute THEN
				usiTemp						:= ncINC_OUTPUT;

				fbWriteParID.Axis			:= ADR(i_pstEncEmulAxis);
				fbWriteParID.DataAddress 	:= ADR(usiTemp);
				fbWriteParID.DataType		:= ncPAR_TYP_USINT;
				fbWriteParID.ParID			:= ACP10PAR_ENCOD_TYPE;
				fbWriteParID.Execute		:= TRUE;
			END_IF

			IF fbWriteParID.Done AND fbWriteParID.ParID = ACP10PAR_ENCOD_TYPE THEN
				fbWriteParID.Execute	:= FALSE;
				uiStep					:= 20;
			ELSIF fbWriteParID.Error THEN
				uiStep					:= 900;
			END_IF
		(* ENCODER MODE CONFIG *)
		20:(* INC MODE *)
			IF NOT fbWriteParID.Execute THEN
				uiTemp						:= 4;

				fbWriteParID.Axis			:= ADR(i_pstEncEmulAxis);
				fbWriteParID.DataAddress 	:= ADR(uiTemp);
				fbWriteParID.DataType		:= ncPAR_TYP_UINT;
				fbWriteParID.ParID			:= ACP10PAR_ENCOD_INC_MODE;
				fbWriteParID.Execute		:= TRUE;
			END_IF

			IF fbWriteParID.Done AND fbWriteParID.ParID = ACP10PAR_ENCOD_INC_MODE THEN
				fbWriteParID.Execute	:= FALSE;
				uiStep					:= 30;
			ELSIF fbWriteParID.Error THEN
				uiStep					:= 900;
			END_IF

		30:(* SCALE ENC INCREMENT CONFIG *)
			IF NOT fbWriteParID.Execute THEN
				udiTemp						:= UINT_TO_UDINT(i_uiNumberOfPulses) * 64;

				fbWriteParID.Axis			:= ADR(i_pstEncEmulAxis);
				fbWriteParID.DataAddress 	:= ADR(udiTemp);
				fbWriteParID.DataType		:= ncPAR_TYP_UDINT;
				fbWriteParID.ParID			:= ACP10PAR_SCALE_ENCOD_INCR;
				fbWriteParID.Execute		:= TRUE;
			END_IF

			IF fbWriteParID.Done AND fbWriteParID.ParID = ACP10PAR_SCALE_ENCOD_INCR THEN
				fbWriteParID.Execute	:= FALSE;
				uiStep					:= 40;
			ELSIF fbWriteParID.Error THEN
				uiStep					:= 900;
			END_IF

		40:(* SCALE LOAD UNITS CONFIG *)
			IF NOT fbWriteParID.Execute THEN
				udiTemp						:= 36000;

				fbWriteParID.Axis			:= ADR(i_pstEncEmulAxis);
				fbWriteParID.DataAddress 	:= ADR(udiTemp);
				fbWriteParID.DataType		:= ncPAR_TYP_UDINT;
				fbWriteParID.ParID			:= ACP10PAR_SCALE_LOAD_UNITS;
				fbWriteParID.Execute		:= TRUE;
			END_IF

			IF fbWriteParID.Done AND fbWriteParID.ParID = ACP10PAR_SCALE_LOAD_UNITS THEN
				fbWriteParID.Execute	:= FALSE;
				IF i_pstSrcAxis.nc_obj_inf.node_nr = i_pstEncEmulAxis.nc_obj_inf.node_nr THEN
					uiStep := 200;		//CONFIGURE CROSSLINK
				ELSE
					uiStep := 100;		//CONFIGURE NETWORK COUPLING
				END_IF
			ELSIF fbWriteParID.Error THEN
				uiStep := 900;
			END_IF

		(************************** CONFIGURE NETWORK COUPLING ******************************)
		100:(* Sender config: MA3_CYCLIC_SEND <- PCTRL_S_SET / S_VAX1 *)
			IF NOT fbWriteParID.Execute THEN
				IF i_pstSrcAxis.nc_obj_inf.nc_obj_typ = ncAXIS THEN
					uiTemp		:= ACP10PAR_PCTRL_S_SET; 	//REAL AXIS
				ELSE
					uiTemp		:= ACP10PAR_S_SET_VAX1;		//VIRTUAL AXIS
				END_IF

				fbWriteParID.Axis			:= ADR(i_pstSrcAxis);
				fbWriteParID.DataAddress 	:= ADR(uiTemp);
				fbWriteParID.DataType		:= ncPAR_TYP_UINT;
				fbWriteParID.ParID			:= ACP10PAR_MA3_CYCLIC_SEND;
				fbWriteParID.Execute		:= TRUE;
			END_IF

			IF fbWriteParID.Done AND fbWriteParID.ParID = ACP10PAR_MA3_CYCLIC_SEND THEN
				fbWriteParID.Execute	:= FALSE;
				uiStep					:= 120;
			ELSIF fbWriteParID.Error THEN
				uiStep					:= 900;
			END_IF

		120:(* Receiver config : MA5_CYCLIC_POS <- "node_nr [+ 256 for AXIS 2], MA3_CYCLIC_SEND" *)
			IF NOT fbWriteParID_Text.Execute THEN
				uiTemp		:= i_pstSrcAxis.nc_obj_inf.node_nr + 256 * (i_pstSrcAxis.nc_obj_inf.nc_obj_idx);
				itoa(uiTemp, ADR(strTemp));
				uiTemp		:= ACP10PAR_MA3_CYCLIC_SEND;
				itoa(uiTemp, ADR(strTemp2));

				strcat(ADR(strTemp), ADR(', '));
				strcat(ADR(strTemp), ADR(strTemp2));

				fbWriteParID_Text.Axis			:= ADR(i_pstEncEmulAxis);
				fbWriteParID_Text.DataText	 	:= strTemp;
				fbWriteParID_Text.ParID			:= ACP10PAR_CONFIG_MA5_CYCLIC_POS;
				fbWriteParID_Text.Execute		:= TRUE;
			END_IF

			IF fbWriteParID_Text.Done AND fbWriteParID_Text.ParID = ACP10PAR_CONFIG_MA5_CYCLIC_POS THEN
				fbWriteParID_Text.Execute	:= FALSE;
				uiStep						:= 140;
			ELSIF fbWriteParID_Text.Error THEN
				uiStep					:= 900;
			END_IF

		140:(* Set interpolation mode = LINEAR *)
			IF NOT fbWriteParID.Execute THEN
				usiTemp						:= 1;	//LINEAR MODE

				fbWriteParID.Axis			:= ADR(i_pstEncEmulAxis);
				fbWriteParID.DataAddress 	:= ADR(usiTemp);
				fbWriteParID.DataType		:= ncPAR_TYP_USINT;
				fbWriteParID.ParID			:= ACP10PAR_MA5_CYCLIC_IPL_MODE;
				fbWriteParID.Execute		:= TRUE;
			END_IF

			IF fbWriteParID.Done AND fbWriteParID.ParID = ACP10PAR_MA5_CYCLIC_IPL_MODE THEN
				fbWriteParID.Execute	:= FALSE;
				uiStep					:= 150;
			ELSIF fbWriteParID.Error THEN
				uiStep					:= 900;
			END_IF

		150:(* CHECK COMMUNICATION STATUS *)
			IF NOT fbReadParID.Execute THEN
				fbReadParID.Axis			:= ADR(i_pstEncEmulAxis);
				fbReadParID.DataAddress 	:= ADR(usiErrCode);
				fbReadParID.DataType		:= ncPAR_TYP_USINT;
				fbReadParID.ParID			:= ACP10PAR_MA5_CYCLIC_ERROR_STATUS;
				fbReadParID.Execute			:= TRUE;
			END_IF

			IF fbReadParID.Done AND fbReadParID.ParID = ACP10PAR_MA5_CYCLIC_ERROR_STATUS THEN
				fbReadParID.Execute	:= FALSE;
				IF usiErrCode = ERR_OK THEN
					uiEncodOutParID		:= ACP10PAR_MA5_CYCLIC_POS;
					IF i_xEnable THEN
						uiStep	:= 250;
					ELSE
						uiStep	:= 400;
					END_IF
				ELSE
					uiStep				:= 800;
				END_IF
			ELSIF fbReadParID.Error THEN
				uiStep					:= 900;
			END_IF

		(**************************** CONFIGURE CROSSLINK ****************************)
		200:(* CONFIGURE CROSSLINK SOURCE AXIS *)
			IF NOT fbWriteParID.Execute THEN
				uiTemp						:= i_pstSrcAxis.nc_obj_inf.nc_obj_idx + 1;

				fbWriteParID.Axis			:= ADR(i_pstEncEmulAxis);
				fbWriteParID.DataAddress 	:= ADR(uiTemp);
				fbWriteParID.DataType		:= ncPAR_TYP_UINT;
				fbWriteParID.ParID			:= ACP10PAR_CROSSLINK_AXIS;
				fbWriteParID.Execute		:= TRUE;
			END_IF

			IF fbWriteParID.Done AND fbWriteParID.ParID = ACP10PAR_CROSSLINK_AXIS THEN
				fbWriteParID.Execute	:= FALSE;
				uiStep					:= 210;
			ELSIF fbWriteParID.Error THEN
				uiStep					:= 900;
			END_IF

		210:(* CONFIGURE CROSSLINK PARID <- PCTRL_S_SET / S_SET_VAX1 *)
			IF NOT fbWriteParID.Execute THEN
				IF i_pstSrcAxis.nc_obj_inf.nc_obj_typ = ncAXIS THEN
					uiTemp		:= ACP10PAR_PCTRL_S_SET;	//REAL AXIS
				ELSE
					uiTemp		:= ACP10PAR_S_SET_VAX1;		//VIRTUAL AXIS
				END_IF

				fbWriteParID.Axis			:= ADR(i_pstEncEmulAxis);
				fbWriteParID.DataAddress 	:= ADR(uiTemp);
				fbWriteParID.DataType		:= ncPAR_TYP_UINT;
				fbWriteParID.ParID			:= ACP10PAR_CROSSLINK_PARID;
				fbWriteParID.Execute		:= TRUE;
			END_IF

			IF fbWriteParID.Done AND fbWriteParID.ParID = ACP10PAR_CROSSLINK_PARID THEN
				fbWriteParID.Execute	:= FALSE;
				uiEncodOutParID			:= ACP10PAR_CROSSLINK_PARID;
				IF i_xEnable THEN
					uiStep	:= 250;
				ELSE
					uiStep	:= 400;
				END_IF
			ELSIF fbWriteParID.Error THEN
				uiStep					:= 900;
			END_IF

		250:(* ENABLE ENCODER EMULATOR OUTPUT *)
			IF NOT fbWriteParID.Execute THEN
				fbWriteParID.Axis			:= ADR(i_pstEncEmulAxis);
				fbWriteParID.DataAddress 	:= ADR(uiEncodOutParID);
				fbWriteParID.DataType		:= ncPAR_TYP_UINT;
				fbWriteParID.ParID			:= ACP10PAR_ENCOD_OUT_PARID;
				fbWriteParID.Execute		:= TRUE;
			END_IF

			IF fbWriteParID.Done AND fbWriteParID.ParID = ACP10PAR_ENCOD_OUT_PARID THEN
				fbWriteParID.Execute	:= FALSE;
				uiStep					:= 300;
			ELSIF fbWriteParID.Error THEN
				uiStep					:= 900;
			END_IF

		300:(* READY *)
			fbAxisError.Enable	:= TRUE;
			q_xActive			:= TRUE;

			IF NOT i_xEnable THEN
				uiStep			:= 400;
			END_IF

		400:(* DISABLE OUTPUT *)
			//fbAxisError.Enable	:= FALSE; //V4.A.A.1.6.13

			IF NOT fbWriteParID.Execute THEN
				uiTemp						:= 0;

				fbWriteParID.Axis			:= ADR(i_pstEncEmulAxis);
				fbWriteParID.DataAddress 	:= ADR(uiTemp);
				fbWriteParID.DataType		:= ncPAR_TYP_UINT;
				fbWriteParID.ParID			:= ACP10PAR_ENCOD_OUT_PARID;
				fbWriteParID.Execute		:= TRUE;
			END_IF

			IF fbWriteParID.Done AND fbWriteParID.ParID = ACP10PAR_ENCOD_OUT_PARID THEN
				fbWriteParID.Execute	:= FALSE;
				q_xActive 				:= FALSE;
				uiStep	:= 410;
			END_IF

		410: (* OUTPUT DISABLED *)
			IF i_xEnable THEN
				uiStep	:= 250;
			END_IF

		(********************************************)
		800:(* CYCLIC COMMUNICATION ERROR *)
			q_xError 		:= TRUE;
			q_uiErrorID		:= usiErrCode;
			IF i_xErrorReset THEN
				q_xError 	:= FALSE;
				q_uiErrorID := 0;
				uiStep		:= 0;
			END_IF

		900:(* FUNCTION BLOCKS ERROR *)
			q_xError 		:= TRUE;
			q_uiErrorID 	:= fbWriteParID.ErrorID + fbReadParID.ErrorID + fbWriteParID_Text.ErrorID;

			fbWriteParID.Execute 	:= FALSE;
			fbReadParID.Execute 	:= FALSE;

			IF i_xErrorReset THEN
				IF fbWriteParID.Error THEN
					fbWriteParID.Execute := FALSE;
				END_IF
				IF fbReadParID.Error THEN
					fbReadParID.Execute := FALSE;
				END_IF
				IF fbWriteParID_Text.Error THEN
					fbReadParID.Execute := FALSE;
				END_IF
			END_IF

			IF NOT fbWriteParID.Error AND NOT fbReadParID.Error AND NOT fbWriteParID_Text.Error THEN
				q_xError 		:= FALSE;
				q_uiErrorID 	:= 0;
				uiStep			:= 0;
			END_IF

		950:
			fbWriteParID.Execute 	:= FALSE;
			fbReadParID.Execute 	:= FALSE;

			q_xError 		:= TRUE;
			q_uiErrorID		:= 60000;
			IF i_pstEncEmulAxis.network.phase  = 90 THEN
				uiStep	:= 0;
			END_IF

		960:
			fbWriteParID.Execute 	:= FALSE;
			fbReadParID.Execute 	:= FALSE;

			q_xError 	:= TRUE;
			q_uiErrorID	:= 60010;

			IF i_xErrorReset THEN
				fbAxisError.Enable	:= FALSE;
			END_IF

			IF NOT fbAxisError.Error THEN
				uiStep	:= 0;
			END_IF

		970:
			q_xError 	:= TRUE;
			q_uiErrorID	:= 60020;

			fbWriteParID.Execute 	:= FALSE;
			fbReadParID.Execute 	:= FALSE;

			//fbAxisError.Acknowledge	:= i_xErrorReset; //V4.A.A.1.6.13

			IF NOT(fbAxisError.FunctionBlockErrorCount > 0 OR fbAxisError.AxisErrorCount > 0) THEN
				//fbAxisError.Enable	:= FALSE; //V4.A.A.1.6.13
				uiStep	:= 0;
			END_IF
	END_CASE

	(* Acknowledge Error *)
	fbAxisError.Acknowledge	:= i_xErrorReset;

	fbAxisError();
	fbReadParID();
	fbWriteParID_Text();
	fbWriteParID();
END_FUNCTION_BLOCK
```

#### FB_CamGeneratorAB.st
```iecst
(* Cam Generator Function Block *)
FUNCTION_BLOCK FB_CamGeneratorAB
	IF i_xEnable THEN
		IF (i_rOnPositionA <> i_rOffPositionA) AND (i_rOnPositionB <> i_rOffPositionB) THEN
			rAdvPosition		:= i_rAdvanceTime * i_prAxisVelocity / 1000.0;
			q_xAdvError			:= (ABS(rAdvPosition) >= 360);

			i_pxPointerStepAdvA	:= ((i_rOnPositionA - rAdvPosition) < 0);
			i_pxPointerStepAdvB	:= ((i_rOnPositionB - rAdvPosition) < 0);

			rOnPositionA		:= FC_RealReminder(i_rOnPositionA - rAdvPosition,	360.0, 0);
			rOffPositionA		:= FC_RealReminder(i_rOffPositionA - rAdvPosition,	360.0, 0);

			rOnPositionB		:= FC_RealReminder(i_rOnPositionB - rAdvPosition,	360.0, 0);
			rOffPositionB		:= FC_RealReminder(i_rOffPositionB - rAdvPosition,	360.0, 0);

			(* CAM A GENERATION *)
			IF(rOnPositionA < rOffPositionA) THEN
				xCamValueA	:= (i_plrAxisPosition >= rOnPositionA) AND (i_plrAxisPosition < rOffPositionA);
			ELSE
				xCamValueA	:= i_plrAxisPosition >= rOnPositionA OR i_plrAxisPosition < rOffPositionA;
			END_IF

			IF xCamValueA <> xOldCamValueA THEN
				rTempReal	:= SEL(xCamValueA, rOffPositionA, rOnPositionA);
				rTempReal	:= rTempReal - LREAL_TO_REAL(i_plrAxisPosition);
				IF ABS(rTempReal) > 0.5 AND ABS(rTempReal) < 359.5 THEN
					xOldCamValueA := xCamValueA;
				END_IF
			END_IF

			(* CAM B GENERATION *)
			IF(rOnPositionB < rOffPositionB) THEN
				xCamValueB	:= (i_plrAxisPosition >= rOnPositionB) AND (i_plrAxisPosition < rOffPositionB);
			ELSE
				xCamValueB	:= i_plrAxisPosition >= rOnPositionB OR i_plrAxisPosition < rOffPositionB;
			END_IF

			IF xCamValueB <> xOldCamValueB THEN
				rTempReal	:= SEL(xCamValueB, rOffPositionB, rOnPositionB);
				rTempReal	:= rTempReal - LREAL_TO_REAL(i_plrAxisPosition);
				IF ABS(rTempReal) > 0.5 AND ABS(rTempReal) < 359.5 THEN
					xOldCamValueB	:=	xCamValueB;
				END_IF
			END_IF

			(* Debounce *)
			CASE usiStep OF
				0:(* INIT *)
					usiStep := 10;

				10:(* WAIT FIRST CAM RAISING EDGE *)
					IF rOnPositionB < rOffPositionA THEN
						IF xCamValueA THEN
							i_pxPointerOutputA := TRUE;
							usiStep := 100;
						END_IF
					ELSE
						IF xCamValueB THEN
							i_pxPointerOutputB := TRUE;
							usiStep := 200;
						END_IF
					END_IF

				100:(* WAIT CAM B RISE EDGE *)
					IF xCamValueB THEN
						i_pxPointerOutputB := TRUE;
						usiStep := 110;
					END_IF

				110:(* WAIT CAM A FALLING EDGE *)
					IF NOT xCamValueA THEN
						i_pxPointerOutputA := FALSE;
						usiStep := 120;
					END_IF

				120:(* WAIT FOR CAM B FALLING EDGE *)
					IF NOT xCamValueB THEN
						i_pxPointerOutputB := FALSE;
						usiStep := 10;
					END_IF

				200:(* WAIT CAM A RISE EDGE *)
					IF xCamValueA THEN
						i_pxPointerOutputA := TRUE;
						usiStep := 210;
					END_IF

				210:(* WAIT CAM B FALLING EDGE *)
					IF NOT xCamValueB THEN
						i_pxPointerOutputB := FALSE;
						usiStep := 220;
					END_IF

				220:(* WAIT FOR CAM A FALLING EDGE *)
					IF NOT xCamValueA THEN
						i_pxPointerOutputA := FALSE;
						usiStep := 10;
					END_IF

				ELSE
					usiStep := 255;
			END_CASE
		END_IF
	ELSE
		i_pxPointerOutputA	:= FALSE;
		i_pxPointerOutputB	:= FALSE;
		q_xAdvError			:= FALSE;
	END_IF
END_FUNCTION_BLOCK

(* Cam Generator Function Block *)
FUNCTION_BLOCK FB_CamGeneratorAB_v2
	IF i_xEnable THEN
		IF (i_rOnPositionA <> i_rOffPositionA) AND (i_rOnPositionB <> i_rOffPositionB) THEN
			rPosition			:= DINT_TO_REAL(i_pdiAxisPosition MOD 36000) / 100.0;
			rAdvPosition		:= i_rAdvanceTime * i_prAxisVelocity / 100000.0; //v1.6
			q_xAdvError			:= (ABS(rAdvPosition) >= 360);

			i_pxPointerStepAdvA	:= ((i_rOnPositionA - rAdvPosition) < 0);
			i_pxPointerStepAdvB	:= ((i_rOnPositionB - rAdvPosition) < 0);

			rOnPositionA		:= FC_RealReminder(i_rOnPositionA - rAdvPosition,	360.0, 0);
			rOffPositionA		:= FC_RealReminder(i_rOffPositionA - rAdvPosition,	360.0, 0);

			rOnPositionB		:= FC_RealReminder(i_rOnPositionB - rAdvPosition,	360.0, 0);
			rOffPositionB		:= FC_RealReminder(i_rOffPositionB - rAdvPosition,	360.0, 0);

			(* CAM A GENERATION *)
			IF(rOnPositionA < rOffPositionA) THEN
				xCamValueA	:= (rPosition >= rOnPositionA) AND (rPosition < rOffPositionA);
			ELSE
				xCamValueA	:= rPosition >= rOnPositionA OR rPosition < rOffPositionA;
			END_IF

			IF xCamValueA <> xOldCamValueA THEN
				rTempReal	:= SEL(xCamValueA, rOffPositionA, rOnPositionA);
				rTempReal	:= rTempReal - rPosition;
				IF ABS(rTempReal) > 0.5 AND ABS(rTempReal) < 359.5 THEN
					xOldCamValueA := xCamValueA;
				END_IF
			END_IF

			(* CAM B GENERATION *)
			IF(rOnPositionB < rOffPositionB) THEN
				xCamValueB	:= (rPosition >= rOnPositionB) AND (rPosition < rOffPositionB);
			ELSE
				xCamValueB	:= rPosition >= rOnPositionB OR rPosition < rOffPositionB;
			END_IF

			IF xCamValueB <> xOldCamValueB THEN
				rTempReal	:= SEL(xCamValueB, rOffPositionB, rOnPositionB);
				rTempReal	:= rTempReal - rPosition;
				IF ABS(rTempReal) > 0.5 AND ABS(rTempReal) < 359.5 THEN
					xOldCamValueB	:=	xCamValueB;
				END_IF
			END_IF

			(* Debounce *)
			CASE usiStep OF
				0:(* INIT *)
					usiStep := 10;

				10:(* WAIT FIRST CAM RAISING EDGE *)
					IF rOnPositionB < rOffPositionA THEN
						IF xCamValueA THEN
							i_pxPointerOutputA := TRUE;
							usiStep := 100;
						END_IF
					ELSE
						IF xCamValueB THEN
							i_pxPointerOutputB := TRUE;
							usiStep := 200;
						END_IF
					END_IF

				100:(* WAIT CAM B RISE EDGE *)
					IF xCamValueB THEN
						i_pxPointerOutputB := TRUE;
						usiStep := 110;
					END_IF

				110:(* WAIT CAM A FALLING EDGE *)
					IF NOT xCamValueA THEN
						i_pxPointerOutputA := FALSE;
						usiStep := 120;
					END_IF

				120:(* WAIT FOR CAM B FALLING EDGE *)
					IF NOT xCamValueB THEN
						i_pxPointerOutputB := FALSE;
						usiStep := 10;
					END_IF

				200:(* WAIT CAM A RISE EDGE *)
					IF xCamValueA THEN
						i_pxPointerOutputA := TRUE;
						usiStep := 210;
					END_IF

				210:(* WAIT CAM B FALLING EDGE *)
					IF NOT xCamValueB THEN
						i_pxPointerOutputB := FALSE;
						usiStep := 220;
					END_IF

				220:(* WAIT FOR CAM A FALLING EDGE *)
					IF NOT xCamValueA THEN
						i_pxPointerOutputA := FALSE;
						usiStep := 10;
					END_IF

				ELSE
					usiStep := 255;
			END_CASE
		END_IF
	ELSE
		i_pxPointerOutputA	:= FALSE;
		i_pxPointerOutputB	:= FALSE;
		q_xAdvError			:= FALSE;
	END_IF
END_FUNCTION_BLOCK
```

#### FB_DigitalCam.st
```iecst
FUNCTION_BLOCK FB_DigitalCam
	IF i_rOnCam > 360.0 OR i_rOnCam < 0.0 OR i_rOffCam > 360.0 OR i_rOffCam < 0.0 THEN
		uiMngStep	:= 9999;
	END_IF

	IF ((i_rOnCam = i_rOffCam) AND (i_usiPulses <= 1)) OR (i_usiPulses = 0) THEN
		uiMngStep := 0;
	END_IF

	IF i_pstAxis.move.mode <> ncPAR_LIST_MOVE AND uiMngStep = 100 AND fbCamSwitch.Enable THEN
		uiMngStep := 10;
	END_IF

	CASE uiMngStep OF
		0: 	(* Idle - Check parameters consistation *)
			fbCamSwitch.InitTrackOptions	:= FALSE;
			fbCamSwitch.Enable				:= FALSE;

			IF (i_rOnCam <> i_rOffCam) OR (i_usiPulses > 1) THEN
				uiMngStep := 100;
				stMasterSwitch.Master	:= ADR(i_pstAxis);
				stMasterSwitch.Period 	:= 360.0;
			END_IF

		10:
			fbCamSwitch.InitTrackOptions	:= FALSE;
			fbCamSwitch.Enable				:= FALSE;

			IF i_pstAxis.move.mode = ncPAR_LIST_MOVE THEN
				uiMngStep := 100;
				fbCamSwitch.Enable	:= TRUE;
			END_IF

		100:
			IF EDGEPOS(i_xRefreshClock) THEN
				IF usiMultiPulse <> i_usiPulses THEN
					uiMngStep := 600;
				ELSIF usiMultiPulse = 1 THEN
					IF stMasterSwitch.MasterStartPosition = 0.0 THEN
						IF (i_rOnCam <> stMasterSwitch.Switches[0].FirstOnPosition[0]) OR
							(i_rOffCam <> stMasterSwitch.Switches[0].LastOnPosition[0]) THEN
							stMasterSwitch.Switches[0].FirstOnPosition[0]	:= i_rOnCam;
							stMasterSwitch.Switches[0].LastOnPosition[0]	:= i_rOffCam;
							uiMngStep := 500;
						END_IF
					ELSE
						IF (i_rOnCam <> stMasterSwitch.MasterStartPosition) OR
							(i_rOffCam <> (stMasterSwitch.Switches[0].LastOnPosition[0] - (360.0 - stMasterSwitch.MasterStartPosition))) THEN
							stMasterSwitch.Switches[0].FirstOnPosition[0]	:= i_rOnCam;
							stMasterSwitch.Switches[0].LastOnPosition[0]	:= i_rOffCam;
							uiMngStep := 500;
						END_IF
					END_IF
				ELSIF i_rAdvTime <> (stTrackOption.OnCompensation * 1000.0) THEN
					uiMngStep := 400;
				END_IF
			END_IF

		400:
			stTrackOption.OnCompensation	:= i_rAdvTime / 1000.0;
			stTrackOption.OffCompensation	:= i_rAdvTime / 1000.0;
			fbCamSwitch.InitTrackOptions	:= TRUE;
			uiMngStep := 410;

		410:
			IF fbCamSwitch.TrackOptionsInitialized THEN
				fbCamSwitch.InitTrackOptions	:= FALSE;
				uiMngStep := 100;
			END_IF

		500:	(* Check parameters consistation *)
			IF stMasterSwitch.Switches[0].FirstOnPosition[0] < stMasterSwitch.Switches[0].LastOnPosition[0] THEN
				uiMngStep := 700;
			ELSE
				uiMngStep := 800;
			END_IF

		600:
			FOR usiTemp := 0 TO MAX(usiMultiPulse, i_usiPulses) - 1 DO
				IF usiTemp <= i_usiPulses - 1 THEN
					IF usiTemp = 0 THEN
						stMasterSwitch.Switches[0].FirstOnPosition[usiTemp]	:= 0.0;
						stMasterSwitch.Switches[0].LastOnPosition[usiTemp]	:= 180.0 / USINT_TO_REAL(i_usiPulses);
					ELSE
						stMasterSwitch.Switches[0].FirstOnPosition[usiTemp]	:= stMasterSwitch.Switches[0].LastOnPosition[0] * USINT_TO_REAL(usiTemp * 2);
						stMasterSwitch.Switches[0].LastOnPosition[usiTemp]	:= stMasterSwitch.Switches[0].LastOnPosition[0] * (USINT_TO_REAL(usiTemp * 2) + 1.0);
					END_IF
				ELSE
					stMasterSwitch.Switches[0].FirstOnPosition[usiTemp]	:= 0.0;
					stMasterSwitch.Switches[0].LastOnPosition[usiTemp]	:= 0.0;
				END_IF
			END_FOR

			usiMultiPulse := i_usiPulses;
			stMasterSwitch.MasterStartPosition	:= 0.0;
			stTrackOption.OnCompensation		:= i_rAdvTime / 1000.0;
			stTrackOption.OffCompensation		:= i_rAdvTime / 1000.0;
			uiMngStep := 2000;

		700:	(* Init switch 4 *)
			stMasterSwitch.MasterStartPosition	:= 0.0;
			stTrackOption.OnCompensation		:= i_rAdvTime / 1000.0;
			stTrackOption.OffCompensation		:= i_rAdvTime / 1000.0;
			uiMngStep := 2000;

		800:
			stMasterSwitch.MasterStartPosition				:= stMasterSwitch.Switches[0].FirstOnPosition[0];
			stMasterSwitch.Switches[0].LastOnPosition[0]	:= stMasterSwitch.Switches[0].LastOnPosition[0] + (360.0 - stMasterSwitch.Switches[0].FirstOnPosition[0]);
			stMasterSwitch.Switches[0].FirstOnPosition[0]	:= 0.0;
			stTrackOption.OnCompensation					:= i_rAdvTime / 1000.0;
			stTrackOption.OffCompensation					:= i_rAdvTime / 1000.0;
			uiMngStep := 2000;

		2000:
			IF EDGENEG(fbCamSwitch.Value) OR NOT fbCamSwitch.Enable THEN
				fbCamSwitch.Enable	:= FALSE;
				uiMngStep		:= 2010;
			END_IF

		2010:
			IF NOT fbCamSwitch.InOperation THEN
				fbCamSwitch.Enable	:= TRUE;
				uiMngStep		:= 2020;
			END_IF

		2020:
			IF NOT fbCamSwitch.Error AND fbCamSwitch.InOperation THEN
				uiMngStep := 100;
				xCamInitialized := TRUE;
			END_IF

		9999:
			IF NOT(i_rOnCam > 360.0 OR i_rOnCam > 0.0 OR i_rOffCam > 360.0 OR i_rOffCam > 0.0) THEN
				uiMngStep	:= 0;
			END_IF
	END_CASE

	fbCamSwitch(
	Switches		:= stMasterSwitch,
	OutputOptions	:= stOutputOption,
	TrackOptions	:= stTrackOption,
	EnableValue		:= TRUE,
	);

	q_xOutPulse := fbCamSwitch.Value;
END_FUNCTION_BLOCK
```

#### FB_AbsolutePosCalculation.st
```iecst
FUNCTION_BLOCK FB_AbsolutePosCalculation
	IF i_xEnable THEN

		IF NOT i_pstAxis.iq_stStatus.q_stMainAxisStatus.q_xInitDone OR i_pstAxis.iq_stStatus.q_stMainAxisStatus.q_xError THEN
			xPositionValid 		:= FALSE;
		ELSIF i_xPositionSensor AND NOT xPositionValid THEN
			lrAbsolutePosition 	:= i_pstAxis.iq_stStatus.q_stMainAxisStatus.q_lrPosition + 360.0 * MAX((i_uiAbsolutePositionOffset - 1), 0);
			xPositionValid 		:= TRUE;
			lrOldPosition 		:= i_pstAxis.iq_stStatus.q_stMainAxisStatus.q_lrPosition;
		ELSE
			lrIncrement			:= i_pstAxis.iq_stStatus.q_stMainAxisStatus.q_lrPosition - lrOldPosition;

			IF lrIncrement < -180.0 THEN
				lrIncrement := lrIncrement + 360.0;
			ELSIF lrIncrement > 180.0 THEN
				lrIncrement := lrIncrement - 360.0;
			END_IF

			lrAbsolutePosition	:= lrAbsolutePosition + lrIncrement;
			lrOldPosition		:= i_pstAxis.iq_stStatus.q_stMainAxisStatus.q_lrPosition;
		END_IF

		lrAbsolutePosition		:= FC_LongRealReminder(lrAbsolutePosition, 360.0 * i_uiStepsNumber, 0);

		q_xPositionValid		:= xPositionValid;
		q_lrAbsolutePosition	:= lrAbsolutePosition;
	END_IF
END_FUNCTION_BLOCK
```

#### FC_GetAccFromTimeAndJerk.st
```iecst
(* Get the acceleration (deceleration) value from time and jerk *)
FUNCTION FC_GetAccFromTimeAndJerk
	IF i_rTime = 0 THEN
		rTime := 20;
	ELSE
		rTime := i_rTime;
	END_IF

	IF i_rVelocity <= 0 THEN
		FC_GetAccFromTimeAndJerk :=	500;
		RETURN;
	END_IF

	IF i_rJerk <= 0 THEN
		FC_GetAccFromTimeAndJerk :=	i_rVelocity	/ rTime;
		RETURN;
	ELSE
		rTemp := rTime * rTime - 4 * i_rVelocity / i_rJerk;
		IF rTemp >= 0 THEN
			rTemp := SQRT(rTemp);
			rFistSolution	:= (i_rTime + rTemp) * i_rJerk / 2;
			rSecondSolution	:= (i_rTime - rTemp) * i_rJerk / 2;
			IF i_rVelocity >= (rFistSolution * rFistSolution) / i_rJerk THEN
				FC_GetAccFromTimeAndJerk := rFistSolution;
			ELSIF i_rVelocity >= (rSecondSolution * rSecondSolution) / i_rJerk THEN
				FC_GetAccFromTimeAndJerk := rSecondSolution;
			ELSE
				FC_GetAccFromTimeAndJerk := i_rVelocity / rTime;
			END_IF
		ELSE
			FC_GetAccFromTimeAndJerk :=	i_rVelocity	/ rTime;
		END_IF
	END_IF
END_FUNCTION
```

#### FC_diReminder.st
```iecst
FUNCTION FC_diReminder
	diReminder_a	:= (i_diDividend - (i_diDividend / i_diDivisor) * i_diDivisor);
	diReminder_b	:= (diReminder_a + i_diDivisor - ((diReminder_a + i_diDivisor) / i_diDivisor) * i_diDivisor);

	FC_diReminder	:= (diReminder_b + i_diStart - (((diReminder_b + i_diStart) / i_diDivisor) * i_diDivisor));
END_FUNCTION
```

#### FC_LongRealReminder.st
```iecst
FUNCTION FC_LongRealReminder
	lrReminder_a	:= (i_lrDividend - (DINT_TO_LREAL(TRUNC(i_lrDividend / i_lrDivisor)) * i_lrDivisor));
	lrReminder_b	:= (lrReminder_a + i_lrDivisor - (DINT_TO_LREAL(TRUNC((lrReminder_a + i_lrDivisor) / i_lrDivisor)) * i_lrDivisor));

	FC_LongRealReminder	:= (lrReminder_b + i_lrStart - (DINT_TO_LREAL(TRUNC((lrReminder_b + i_lrStart) / i_lrDivisor)) * i_lrDivisor));
END_FUNCTION
```

#### FC_RealReminder.st
```iecst
FUNCTION FC_RealReminder
	rReminder_a	:= (i_rDividend - (DINT_TO_REAL(TRUNC(i_rDividend / i_rDivisor)) * i_rDivisor));
	rReminder_b	:= (rReminder_a + i_rDivisor - (DINT_TO_REAL(TRUNC((rReminder_a + i_rDivisor) / i_rDivisor)) * i_rDivisor));

	FC_RealReminder	:= (rReminder_b + i_rStart - (DINT_TO_REAL(TRUNC((rReminder_b + i_rStart) / i_rDivisor)) * i_rDivisor));
END_FUNCTION
```

#### FC_mmToDegree.st
```iecst
FUNCTION FC_mmToDegree
	rTempStep	:= i_rPositionMm * 360.0 / LREAL_TO_REAL(i_lrMachineStep);

	FC_mmToDegree	:= FC_RealReminder(i_rDividend := rTempStep, i_rDivisor := 360.0, i_rStart := 0);
END_FUNCTION
```

#### FC_DegreeToMm.st
```iecst
FUNCTION FC_DegreeToMm
	rTempStep	:= i_rPositionDegree * LREAL_TO_REAL(i_lrMachineStep) / 360.0;

	IF i_xRemindResult THEN
		FC_DegreeToMm	:= FC_RealReminder(i_rDividend := rTempStep, i_rDivisor := LREAL_TO_REAL(i_lrMachineStep), i_rStart := 0);
	ELSE
		FC_DegreeToMm	:= rTempStep;
	END_IF
END_FUNCTION
```

#### FC_TeensOfmmToDegrees.st
```iecst
FUNCTION FC_TeensOfmmToDegrees
	lrTempStep	:= i_iTeensOfmm * 360.0 / (i_lrMachineStep * 10.0);

	IF i_xWithoutModulo THEN
		FC_TeensOfmmToDegrees := lrTempStep;
	ELSIF i_xNegativeResult THEN
		IF lrTempStep >= 0 THEN
			FC_TeensOfmmToDegrees := FC_LongRealReminder(i_lrDividend := lrTempStep, i_lrDivisor:= 360.0, i_lrStart := 0);
		ELSE
			FC_TeensOfmmToDegrees := FC_LongRealReminder(i_lrDividend := lrTempStep, i_lrDivisor := 360.0, i_lrStart := 0) - 360.0;
		END_IF
	ELSE
		FC_TeensOfmmToDegrees := FC_LongRealReminder(i_lrDividend := lrTempStep, i_lrDivisor := 360.0, i_lrStart:= 0);
	END_IF
END_FUNCTION
```

#### FC_RephasingMachine.st
```iecst
(* Function for finding the machine rephasing position *)
FUNCTION FC_RephasingMachine
	(* Before starting is necessary to load axes on both arrays *)
	udiLastAxisIndex	:= 0;

	FOR udiAxisIndex := 0 TO 30 BY 1 DO
		alrPositions[udiAxisIndex]	:= 0.0;
		auiAxisIndex[udiAxisIndex]	:= 0;
	END_FOR

	FOR udiAxisIndex := 0 TO CST_LastInletModuleAxis BY 1 DO
		IF iq_astInletSubModuleAxis[udiAxisIndex].iq_stStatus.q_stMainAxisStatus.q_xAxisReal 		AND NOT
			iq_astInletSubModuleAxis[udiAxisIndex].iq_stStatus.q_stMainAxisStatus.q_xPowerSupply 	AND NOT
			iq_astInletSubModuleAxis[udiAxisIndex].iq_stStatus.q_stMainAxisStatus.q_xVelocityControl THEN

			alrPositions[udiLastAxisIndex]	:= iq_astInletSubModuleAxis[udiAxisIndex].iq_stStatus.q_stMainAxisStatus.q_lrPosition;
			auiAxisIndex[udiLastAxisIndex]	:= udiAxisIndex + 2000; (* To the axis module axes index 2000 is added *)

			udiLastAxisIndex	:= MIN(udiLastAxisIndex + 1, 30);
		END_IF
	END_FOR

	FOR udiAxisIndex := 0 TO CST_LastFillerModuleAxis BY 1 DO
		IF iq_astFillerSubModuleAxis[udiAxisIndex].iq_stStatus.q_stMainAxisStatus.q_xAxisReal 		AND NOT
			iq_astFillerSubModuleAxis[udiAxisIndex].iq_stStatus.q_stMainAxisStatus.q_xPowerSupply 	AND NOT
			iq_astFillerSubModuleAxis[udiAxisIndex].iq_stStatus.q_stMainAxisStatus.q_xVelocityControl THEN

			alrPositions[udiLastAxisIndex]	:= iq_astFillerSubModuleAxis[udiAxisIndex].iq_stStatus.q_stMainAxisStatus.q_lrPosition;
			auiAxisIndex[udiLastAxisIndex]	:= udiAxisIndex;

			udiLastAxisIndex	:= MIN(udiLastAxisIndex + 1, 30);
		END_IF
	END_FOR

	FOR udiAxisIndex := 0 TO CST_LastOutletModuleAxis BY 1 DO
		IF iq_astOutletSubModuleAxis[udiAxisIndex].iq_stStatus.q_stMainAxisStatus.q_xAxisReal 			AND NOT
			iq_astOutletSubModuleAxis[udiAxisIndex].iq_stStatus.q_stMainAxisStatus.q_xPowerSupply 		AND NOT
			iq_astOutletSubModuleAxis[udiAxisIndex].iq_stStatus.q_stMainAxisStatus.q_xVelocityControl THEN

			alrPositions[udiLastAxisIndex]	:= iq_astOutletSubModuleAxis[udiAxisIndex].iq_stStatus.q_stMainAxisStatus.q_lrPosition;
			auiAxisIndex[udiLastAxisIndex]	:= udiAxisIndex + 1000; (* To the axis module axes index 1000 is added *)

			udiLastAxisIndex	:= MIN(udiLastAxisIndex + 1, 30);
		END_IF
	END_FOR

	IF udiLastAxisIndex > 1 THEN
		FOR udiRowIndex := 0 TO udiLastAxisIndex - 1 BY 1 DO  (* First Step : make the distance between an axis and the other ones *)
			FOR udiColumnIndex := 0 TO udiLastAxisIndex - 1 BY 1 DO
				aalrDistances[udiRowIndex,udiColumnIndex]	:= 0.0;
				IF udiRowIndex <> udiColumnIndex THEN
					aalrDistances[udiRowIndex,udiColumnIndex] := FC_LongRealReminder(i_lrDividend := (alrPositions[udiRowIndex] - alrPositions[udiColumnIndex]),
					i_lrDivisor:= 360.0,
					i_lrStart:= 0.0);
				END_IF
			END_FOR
		END_FOR

		lrMinimumValue	:= 1e100;
		udiAxisIndex	:= 0;

		FOR udiRowIndex := 0 TO udiLastAxisIndex - 1 BY 1 DO (* Second Step. Verify the path of all axes and find the minimum combination *)
			lrTemp	:= 0;
			FOR udiColumnIndex := 0 TO udiLastAxisIndex - 1 BY 1 DO
				IF udiRowIndex <> udiColumnIndex THEN
					lrTemp := aalrDistances[udiRowIndex, udiColumnIndex]	+ lrTemp;
				END_IF
			END_FOR

			IF lrMinimumValue > lrTemp THEN
				udiAxisIndex		:= udiRowIndex;
				lrMinimumValue		:= lrTemp;
			END_IF
		END_FOR

		FC_RephasingMachine := FC_LongRealReminder(i_lrDividend := alrPositions[udiAxisIndex],
													i_lrDivisor:= 360.0,
													i_lrStart:= 0.0);
	ELSE
		FC_RephasingMachine := FC_LongRealReminder(i_lrDividend:= alrPositions[0],
													i_lrDivisor:= 360.0,
													i_lrStart:= 0.0);
	END_IF
END_FUNCTION
```

#### FC_RephasingPositionFiller.st
```iecst
(* Find The Position Of The First Axis *)
FUNCTION FC_RephasingPositionFiller
	FOR udiRowIndex := 0 TO CST_LastFillerModuleAxis BY 1 DO (* First Step : make the distance between an axis and the other ones *)
		FOR udiColumnIndex := 0 TO CST_LastFillerModuleAxis BY 1 DO
			aalrDistances[udiRowIndex, udiColumnIndex]	:= 0.0;
			IF 	udiRowIndex <> udiColumnIndex	AND
				iq_astSubModuleAxis[udiRowIndex].iq_stStatus.q_stMainAxisStatus.q_xAxisReal 				AND
				iq_astSubModuleAxis[udiColumnIndex].iq_stStatus.q_stMainAxisStatus.q_xAxisReal 				AND
				NOT iq_astSubModuleAxis[udiRowIndex].iq_stStatus.q_stMainAxisStatus.q_xPowerSupply 			AND
				NOT iq_astSubModuleAxis[udiColumnIndex].iq_stStatus.q_stMainAxisStatus.q_xPowerSupply 		AND
				NOT iq_astSubModuleAxis[udiRowIndex].iq_stStatus.q_stMainAxisStatus.q_xVelocityControl		AND
				NOT iq_astSubModuleAxis[udiColumnIndex].iq_stStatus.q_stMainAxisStatus.q_xVelocityControl THEN

				aalrDistances[udiRowIndex,udiColumnIndex] := FC_LongRealReminder(i_lrDividend := (iq_astSubModuleAxis[udiRowIndex].iq_stStatus.q_stMainAxisStatus.q_lrPosition - iq_astSubModuleAxis[udiColumnIndex].iq_stStatus.q_stMainAxisStatus.q_lrPosition),
																					i_lrDivisor := 360.0,
																					i_lrStart := 0.0);
			END_IF
		END_FOR
	END_FOR

	lrMinimumValue	:= 1e100;
	udiAxisIndex	:= CST_FirstFillerModuleAxis;

	FOR udiRowIndex := 0 TO CST_LastFillerModuleAxis BY 1 DO (* Second Step. Verify the path of all axes and find the minimum combination *)
		lrTemp	:= 0;
		IF iq_astSubModuleAxis[udiRowIndex].iq_stStatus.q_stMainAxisStatus.q_xAxisReal 			AND
			NOT iq_astSubModuleAxis[udiRowIndex].iq_stStatus.q_stMainAxisStatus.q_xPowerSupply 	AND
			NOT iq_astSubModuleAxis[udiRowIndex].iq_stStatus.q_stMainAxisStatus.q_xVelocityControl THEN

			FOR udiColumnIndex := 0 TO CST_LastFillerModuleAxis BY 1 DO
				IF udiRowIndex <> udiColumnIndex AND
					iq_astSubModuleAxis[udiColumnIndex].iq_stStatus.q_stMainAxisStatus.q_xAxisReal  		AND
					NOT iq_astSubModuleAxis[udiColumnIndex].iq_stStatus.q_stMainAxisStatus.q_xPowerSupply 	AND
					NOT iq_astSubModuleAxis[udiColumnIndex].iq_stStatus.q_stMainAxisStatus.q_xVelocityControl THEN

					lrTemp := aalrDistances[udiRowIndex, udiColumnIndex] + lrTemp;
				END_IF
			END_FOR

			IF lrMinimumValue > lrTemp THEN
				udiAxisIndex		:= udiRowIndex;
				lrMinimumValue		:= lrTemp;
			END_IF
		END_IF
	END_FOR

	FC_RephasingPositionFiller := FC_LongRealReminder(i_lrDividend := iq_astSubModuleAxis[udiAxisIndex].iq_stStatus.q_stMainAxisStatus.q_lrPosition,
														i_lrDivisor := 360.0,
														i_lrStart := 0.0);
END_FUNCTION
```

#### FC_RephasingPositionInlet.st
```iecst
(* Find The Position Of The First Axis *)
FUNCTION FC_RephasingPositionInlet
	FOR udiRowIndex := 0 TO CST_LastInletModuleAxis BY 1 DO (* First Step : make the distance between an axis and the other ones *)
		FOR udiColumnIndex := 0 TO CST_LastInletModuleAxis BY 1 DO
			aalrDistances[udiRowIndex, udiColumnIndex]	:= 0.0;
			IF 	udiRowIndex <> udiColumnIndex	AND
				iq_astSubModuleAxis[udiRowIndex].iq_stStatus.q_stMainAxisStatus.q_xAxisReal 				AND
				iq_astSubModuleAxis[udiColumnIndex].iq_stStatus.q_stMainAxisStatus.q_xAxisReal 				AND
				NOT iq_astSubModuleAxis[udiRowIndex].iq_stStatus.q_stMainAxisStatus.q_xPowerSupply 			AND
				NOT iq_astSubModuleAxis[udiColumnIndex].iq_stStatus.q_stMainAxisStatus.q_xPowerSupply 		AND
				NOT iq_astSubModuleAxis[udiRowIndex].iq_stStatus.q_stMainAxisStatus.q_xVelocityControl		AND
				NOT iq_astSubModuleAxis[udiColumnIndex].iq_stStatus.q_stMainAxisStatus.q_xVelocityControl THEN

				aalrDistances[udiRowIndex,udiColumnIndex] := FC_LongRealReminder(i_lrDividend := (iq_astSubModuleAxis[udiRowIndex].iq_stStatus.q_stMainAxisStatus.q_lrPosition - iq_astSubModuleAxis[udiColumnIndex].iq_stStatus.q_stMainAxisStatus.q_lrPosition),
																				i_lrDivisor := 360.0,
																				i_lrStart := 0.0);
			END_IF
		END_FOR
	END_FOR

	lrMinimumValue	:= 1e100;
	udiAxisIndex	:= CST_FirstInletModuleAxis;

	FOR udiRowIndex := 0 TO CST_LastInletModuleAxis BY 1 DO (* Second Step. Verify the path of all axes and find the minimum combination *)
		lrTemp	:= 0;
		IF iq_astSubModuleAxis[udiRowIndex].iq_stStatus.q_stMainAxisStatus.q_xAxisReal 			AND
			NOT iq_astSubModuleAxis[udiRowIndex].iq_stStatus.q_stMainAxisStatus.q_xPowerSupply 	AND
			NOT iq_astSubModuleAxis[udiRowIndex].iq_stStatus.q_stMainAxisStatus.q_xVelocityControl THEN

			FOR udiColumnIndex := 0 TO CST_LastInletModuleAxis BY 1 DO
				IF udiRowIndex <> udiColumnIndex AND
					iq_astSubModuleAxis[udiColumnIndex].iq_stStatus.q_stMainAxisStatus.q_xAxisReal  		AND
					NOT iq_astSubModuleAxis[udiColumnIndex].iq_stStatus.q_stMainAxisStatus.q_xPowerSupply 	AND
					NOT iq_astSubModuleAxis[udiColumnIndex].iq_stStatus.q_stMainAxisStatus.q_xVelocityControl THEN

					lrTemp := aalrDistances[udiRowIndex, udiColumnIndex] + lrTemp;
				END_IF
			END_FOR

			IF lrMinimumValue > lrTemp THEN
				udiAxisIndex		:= udiRowIndex;
				lrMinimumValue		:= lrTemp;
			END_IF
		END_IF
	END_FOR

	FC_RephasingPositionInlet := FC_LongRealReminder(i_lrDividend := iq_astSubModuleAxis[udiAxisIndex].iq_stStatus.q_stMainAxisStatus.q_lrPosition,
														i_lrDivisor := 360.0,
														i_lrStart := 0.0);
END_FUNCTION
```

#### FC_RephasingPositionOutlet.st
```iecst
(* Find The Position Of The First Axis *)
FUNCTION FC_RephasingPositionOutlet
	FOR udiRowIndex := 0 TO CST_LastOutletModuleAxis BY 1 DO (* First Step : make the distance between an axis and the other ones *)
		FOR udiColumnIndex := 0 TO CST_LastOutletModuleAxis BY 1 DO
			aalrDistances[udiRowIndex, udiColumnIndex]	:= 0.0;
			IF 	udiRowIndex <> udiColumnIndex	AND
				iq_astSubModuleAxis[udiRowIndex].iq_stStatus.q_stMainAxisStatus.q_xAxisReal 				AND
				iq_astSubModuleAxis[udiColumnIndex].iq_stStatus.q_stMainAxisStatus.q_xAxisReal 				AND
				NOT iq_astSubModuleAxis[udiRowIndex].iq_stStatus.q_stMainAxisStatus.q_xPowerSupply 			AND
				NOT iq_astSubModuleAxis[udiColumnIndex].iq_stStatus.q_stMainAxisStatus.q_xPowerSupply 		AND
				NOT iq_astSubModuleAxis[udiRowIndex].iq_stStatus.q_stMainAxisStatus.q_xVelocityControl		AND
				NOT iq_astSubModuleAxis[udiColumnIndex].iq_stStatus.q_stMainAxisStatus.q_xVelocityControl THEN

				aalrDistances[udiRowIndex,udiColumnIndex] := FC_LongRealReminder(i_lrDividend := (iq_astSubModuleAxis[udiRowIndex].iq_stStatus.q_stMainAxisStatus.q_lrPosition - iq_astSubModuleAxis[udiColumnIndex].iq_stStatus.q_stMainAxisStatus.q_lrPosition),
																					i_lrDivisor := 360.0,
																					i_lrStart := 0.0);
			END_IF
		END_FOR
	END_FOR

	lrMinimumValue	:= 1e100;
	udiAxisIndex	:= CST_FirstOutletModuleAxis;

	FOR udiRowIndex := 0 TO CST_LastOutletModuleAxis BY 1 DO (* Second Step. Verify the path of all axes and find the minimum combination *)
		lrTemp	:= 0;
		IF iq_astSubModuleAxis[udiRowIndex].iq_stStatus.q_stMainAxisStatus.q_xAxisReal 			AND
			NOT iq_astSubModuleAxis[udiRowIndex].iq_stStatus.q_stMainAxisStatus.q_xPowerSupply 	AND
			NOT iq_astSubModuleAxis[udiRowIndex].iq_stStatus.q_stMainAxisStatus.q_xVelocityControl THEN

			FOR udiColumnIndex := 0 TO CST_LastOutletModuleAxis BY 1 DO
				IF udiRowIndex <> udiColumnIndex AND
					iq_astSubModuleAxis[udiColumnIndex].iq_stStatus.q_stMainAxisStatus.q_xAxisReal  		AND
					NOT iq_astSubModuleAxis[udiColumnIndex].iq_stStatus.q_stMainAxisStatus.q_xPowerSupply 	AND
					NOT iq_astSubModuleAxis[udiColumnIndex].iq_stStatus.q_stMainAxisStatus.q_xVelocityControl THEN

					lrTemp := aalrDistances[udiRowIndex, udiColumnIndex] + lrTemp;
				END_IF
			END_FOR

			IF lrMinimumValue > lrTemp THEN
				udiAxisIndex		:= udiRowIndex;
				lrMinimumValue		:= lrTemp;
			END_IF
		END_IF
	END_FOR

	FC_RephasingPositionOutlet := FC_LongRealReminder(i_lrDividend := iq_astSubModuleAxis[udiAxisIndex].iq_stStatus.q_stMainAxisStatus.q_lrPosition,
														i_lrDivisor := 360.0,
														i_lrStart := 0.0);
END_FUNCTION
```

### Library Logical/30_MC/Libraries/FiltLib (ANSIC, version 2.00.0) - Filters
Depends on: brsystem

#### FiltLib.var - Exported constants
```iecst
(********************************************************************
 * COPYRIGHT -- Bernecker + Rainer
 ********************************************************************
 * Library: FiltLib
 * File: FiltLib.var
 * Author: passaglial
 * Created: July 16, 2010
 ********************************************************************
 * Constants of library FiltLib
 ********************************************************************)
VAR CONSTANT
	FLTLIB_ER_GET_TASKTIME : UINT := 901; (*Not possible to compute the task class time*)
	FLTLIB_ER_CUT_FREQ_TOO_LOW : UINT := 902; (*Cut Frequency too low*)
	FLTLIB_ER_EXT_TIME_TOO_LOW : UINT := 903; (*Extrapolation time too low*)
	FLTLIB_ER_T1_TOO_LOW : UINT := 904; (*Time constant T1 is too low*)
	FLTLIB_ER_T2_TOO_LOW : UINT := 905; (*Time constant T2 is too low*)
END_VAR
```

#### FiltLib.fun - Exported functions and function blocks
```iecst
(********************************************************************
 * COPYRIGHT -- Bernecker + Rainer
 ********************************************************************
 * Library: FiltLib
 * File: FiltLib.fun
 * Author: passaglial
 * Created: July 16, 2010
 ********************************************************************
 * Functions and function blocks of library FiltLib
 ********************************************************************)

FUNCTION_BLOCK PT2_DINT (*PT2 Filter for DINT source data*)
	VAR_INPUT
		Enable : BOOL; (*Enables FB*)
		T1 : LREAL; (*1st Time constant for the filter [Sec]*)
		T2 : LREAL; (*2nd Time constant for the filter [Sec]*)
		U : DINT; (*Source value*)
	END_VAR
	VAR_OUTPUT
		Busy : BOOL; (*FB is working*)
		Valid : BOOL; (*Filtered value is valid*)
		X : DINT; (*Filtered value *)
		Error : BOOL; (*Error is found*)
		ErrorID : UINT; (*Code for the error*)
	END_VAR
	VAR
		U_old : DINT; (*Previous U*)
		Ts : LREAL; (*Sampling Time (task class time) [Sec]*)
		b0 : LREAL; (*Filter parameter*)
		b1 : LREAL; (*Filter parameter*)
		b2 : LREAL; (*Filter parameter*)
		a1 : LREAL; (*Filter parameter*)
		a2 : LREAL; (*Filter parameter*)
		u0 : LREAL; (*Filter u0*)
		u1 : LREAL; (*Filter u1*)
		u2 : LREAL; (*Filter u2*)
		x0 : LREAL; (*Filter x0*)
		x1 : LREAL; (*Filter x1*)
		x2 : LREAL; (*Filter x2*)
	END_VAR
END_FUNCTION_BLOCK

FUNCTION_BLOCK PT1_DINT (*PT1 Filter for DINT source data*)
	VAR_INPUT
		Enable : BOOL; (*Enables FB*)
		T1 : LREAL; (*Time constant for the filter [Sec]*)
		U : DINT; (*Source value*)
	END_VAR
	VAR_OUTPUT
		Busy : BOOL; (*FB is working*)
		Valid : BOOL; (*Filtered value is valid*)
		X : DINT; (*Filtered value *)
		Error : BOOL; (*Error is found*)
		ErrorID : UINT; (*Code for the error*)
	END_VAR
	VAR
		U_old : DINT; (*Previous U*)
		Ts : LREAL; (*Sampling Time (task class time) [Sec]*)
		b0 : LREAL; (*Filter parameter*)
		b1 : LREAL; (*Filter parameter*)
		a1 : LREAL; (*Filter parameter*)
		u0 : LREAL; (*Filter u0*)
		u1 : LREAL; (*Filter u1*)
		x0 : LREAL; (*Filter x0*)
		x1 : LREAL; (*Filter x1*)
	END_VAR
END_FUNCTION_BLOCK

FUNCTION_BLOCK FDT_DINT (*Generic Transfer function*)
	VAR_INPUT
		Enable : BOOL; (*Enables FB*)
		U : DINT; (*Source value*)
		b0 : LREAL; (*Filter parameter*)
		b1 : LREAL; (*Filter parameter*)
		b2 : LREAL; (*Filter parameter*)
		a1 : LREAL; (*Filter parameter*)
		a2 : LREAL; (*Filter parameter*)
	END_VAR
	VAR_OUTPUT
		Busy : BOOL; (*FB is working*)
		Valid : BOOL; (*Filtered value is valid*)
		X : DINT; (*Filtered value *)
		Error : BOOL; (*Error is found*)
		ErrorID : UINT; (*Code for the error*)
	END_VAR
	VAR
		U_old : DINT; (*Previous U*)
		u0 : LREAL; (*Filter u0*)
		u1 : LREAL; (*Filter u1*)
		u2 : LREAL; (*Filter u2*)
		x0 : LREAL; (*Filter x0*)
		x1 : LREAL; (*Filter x1*)
		x2 : LREAL; (*Filter x2*)
	END_VAR
END_FUNCTION_BLOCK

FUNCTION_BLOCK EXT_DINT (*Extrapolator filter*)
	VAR_INPUT
		Enable : BOOL; (*Enables FB*)
		U : DINT; (*Source value*)
		T_ext : LREAL; (*Extrapolation Time [sec]*)
	END_VAR
	VAR_OUTPUT
		Busy : BOOL; (*FB is working*)
		Valid : BOOL; (*Filtered value is valid*)
		X : DINT; (*Filtered value *)
		Error : BOOL; (*Error is found*)
		ErrorID : UINT; (*Code for the error*)
	END_VAR
	VAR
		Ts : LREAL; (*Sampling Time (task class time) [Sec]*)
		b0 : LREAL; (*Filter parameter*)
		b1 : LREAL; (*Filter parameter*)
		b2 : LREAL; (*Filter parameter*)
		a1 : LREAL; (*Filter parameter*)
		a2 : LREAL; (*Filter parameter*)
		U_old : DINT; (*Previous U*)
		u0 : LREAL; (*Filter u0*)
		u1 : LREAL; (*Filter u1*)
		u2 : LREAL; (*Filter u2*)
		x0 : LREAL; (*Filter x0*)
		x1 : LREAL; (*Filter x1*)
		x2 : LREAL; (*Filter x2*)
	END_VAR
END_FUNCTION_BLOCK
```

#### Filtlib_defines.h
```c
/********************************************************************
 * COPYRIGHT -- Bernecker + Rainer
 ********************************************************************
 * Library: FiltLib
 * File: Filtlib_defines.h
 * Author: passaglial
 * Created: July 23, 2010
 *******************************************************************/
#ifndef _FILTLIB_DEFINES_H
#define _FILTLIB_DEFINES_H

#include <bur/plctypes.h>

#define _MAX_DINT      2147483647.0
#define _MIN_DINT     -2147483648.0
#define _RNG_DINT      4294967296.0
#define _PI            3.141592653589793
#define _MIN_CUT_FREQ  0.001

#endif  /* _FILTLIB_DEFINES_H */
```

#### PT1_DINT.c - PT1 Filter for DINT source data
```c
/********************************************************************
 * COPYRIGHT -- Bernecker + Rainer
 ********************************************************************
 * Library: FiltLib
 * File: PT1_DINT.c
 * Author: passaglial
 * Created: July 16, 2010
 ********************************************************************
 * Implementation of library FiltLib
 ********************************************************************/

#include <bur/plctypes.h>

#ifdef __cplusplus
	extern "C"
	{
#endif

#include "FiltLib.h"
#include "Filtlib_defines.h"

#ifdef __cplusplus
	};
#endif

/* Auxiliary Functions */
static void fnInitPt1Dint(struct PT1_DINT* inst);
static void fnCalcPt1Dint(struct PT1_DINT* inst);

/*PT1 Filter for DINT source data*/
void PT1_DINT(struct PT1_DINT* inst)
{

    if(inst->Enable == 0) /* Not enabled? */
    {
        inst->Busy = 0;
        inst->Valid = 0;
        inst->Error = 0;
        inst->ErrorID = 0;
        inst->X = 0;
        return;
    }
    else if(inst->Busy == 0) /* Just enabled? */
    {
       inst->Busy = 1;
       fnInitPt1Dint(inst);
    }

    /*** FB is enabled ***/

    if(inst->Error != 0)
    {
        inst->Busy = 1;
        inst->Valid = 0;
        return;
    }

    fnCalcPt1Dint(inst);

    inst->Busy = 1;
    inst->Valid = 1;
    return;
}

static void fnInitPt1Dint(struct PT1_DINT* inst)
{
    RTInfo_typ rti;
    double alpha;

    rti.enable = 1;
    RTInfo(&rti);

    if(rti.status != ERR_OK)
    {
        inst->ErrorID = FLTLIB_ER_GET_TASKTIME;
        inst->Error = 1;
        return;
    }

    inst->Ts = (double)rti.cycle_time * 1E-6;

    if(inst->T1 < inst->Ts * 1.5)
    {
        inst->Error = 1;
        inst->ErrorID = FLTLIB_ER_T1_TOO_LOW ;
        return;
    }

    alpha = 2.0 * inst->T1 / inst->Ts;

    inst->b0 = 1 / (1 + alpha);
    inst->b1 = 1 / (1 + alpha);
    inst->a1 = (1 - alpha) / (1 + alpha);

    inst->u0 = (double)inst->U;
    inst->u1 = inst->u0;
    inst->x0 = inst->u0;
    inst->U_old = (long signed int)inst->u0;
    return;
}

static void fnCalcPt1Dint(struct PT1_DINT* inst)
{

    inst->u1 = inst->u0;
    inst->x1 = inst->x0;
    inst->u0 += (double)(inst->U - inst->U_old);
    inst->U_old = inst->U;

    inst->x0 = -(inst->a1 * inst->x1) + (inst->b0 * inst->u0) + (inst->b1 * inst->u1);

    if(inst->x0 > _MAX_DINT)
    {
        inst->x0 -= _RNG_DINT;
        inst->u0 -= _RNG_DINT;
        inst->u1 -= _RNG_DINT;
        inst->x1 -= _RNG_DINT;
    }
    else if(inst->x0 < _MIN_DINT)
    {
        inst->x0 += _RNG_DINT;
        inst->u0 += _RNG_DINT;
        inst->u1 += _RNG_DINT;
        inst->x1 += _RNG_DINT;
    }

    inst->X =(signed long int)inst->x0;

    return;
}
```

#### PT2_DINT.c - PT2 Filter for DINT source data
```c
/********************************************************************
 * COPYRIGHT -- Bernecker + Rainer
 ********************************************************************
 * Library: FiltLib
 * File: PT2_DINT.c
 * Author: passaglial
 * Created: July 23, 2010
 ********************************************************************
 * Implementation of library FiltLib
 ********************************************************************/

#include <bur/plctypes.h>

#ifdef __cplusplus
	extern "C"
	{
#endif

#include "FiltLib.h"
#include "Filtlib_defines.h"

#ifdef __cplusplus
	};
#endif

/* private structure */
struct _pt1_coe_str
{
    double a1;
    double b0;
    double b1;
};

/* Auxiliary Functions */
static void fnInitPt2Dint(struct PT2_DINT* inst);
static void fnCalcPt2Dint(struct PT2_DINT* inst);
static void fnCoeffPt1(struct _pt1_coe_str* coe, double Tf, double Ts);

/*PT2 Filter for DINT source data*/
void PT2_DINT(struct PT2_DINT* inst)
{
    if(inst->Enable == 0) /* Not enabled? */
    {
        inst->Busy = 0;
        inst->Valid = 0;
        inst->Error = 0;
        inst->ErrorID = 0;
        inst->X = 0;
        return;
    }
    else if(inst->Busy == 0) /* Just enabled? */
    {
       inst->Busy = 1;
       fnInitPt2Dint(inst);
    }

    /*** FB is enabled ***/

    if(inst->Error != 0)
    {
        inst->Busy = 1;
        inst->Valid = 0;
        return;
    }

    fnCalcPt2Dint(inst);

    inst->Busy = 1;
    inst->Valid = 1;
    return;

}

static void fnInitPt2Dint(struct PT2_DINT* inst)
{
    RTInfo_typ rti;
    struct _pt1_coe_str f1, f2;

    rti.enable = 1;
    RTInfo(&rti);

    if(rti.status != ERR_OK)
    {
        inst->ErrorID = FLTLIB_ER_GET_TASKTIME;
        inst->Error = 1;
        return;
    }

    inst->Ts = (double)rti.cycle_time * 1E-6;

    if(inst->T1 < inst->Ts * 1.5)
    {
        inst->Error = 1;
        inst->ErrorID = FLTLIB_ER_T1_TOO_LOW ;
        return;
    }
    else if(inst->T2 < inst->Ts * 1.5)
    {
        inst->Error = 1;
        inst->ErrorID = FLTLIB_ER_T2_TOO_LOW ;
        return;
    }

    fnCoeffPt1(&f1, inst->T1, inst->Ts);
    fnCoeffPt1(&f2, inst->T2, inst->Ts);

    inst->b0 =  f1.b0 * f2.b0;
    inst->b1 = (f1.b0 * f2.b1) + (f1.b1 * f2.b0);
    inst->b2 = (f1.b1 * f2.b1);
    inst->a1 =  f2.a1 + f1.a1;
    inst->a2 = (f1.a1 * f2.a1);

    inst->u0 = (double)inst->U;
    inst->u1 = inst->u0;
    inst->x0 = inst->u0;
    inst->x1 = inst->u0;
    inst->U_old = (long signed int)inst->u0;
    return;
}

static void fnCoeffPt1(struct _pt1_coe_str* coe, double Tf, double Ts)
{
    double alpha;

    alpha = 2.0 * Tf / Ts;

    coe->b0 = 1 / (1 + alpha);
    coe->b1 = 1 / (1 + alpha);
    coe->a1 = (1 - alpha) / (1 + alpha);

    return;
}

static void fnCalcPt2Dint(struct PT2_DINT* inst)
{

    inst->x2 = inst->x1;
    inst->x1 = inst->x0;
    inst->u2 = inst->u1;
    inst->u1 = inst->u0;
    inst->u0 += (double)(inst->U - inst->U_old);
    inst->U_old = inst->U;

    inst->x0 = -(inst->a1 * inst->x1) -(inst->a2 * inst->x2)
               +(inst->b0 * inst->u0) +(inst->b1 * inst->u1) +(inst->b2 * inst->u2);

    if(inst->x0 > _MAX_DINT)
    {
        inst->x0 -= _RNG_DINT;
        inst->x1 -= _RNG_DINT;
        inst->x2 -= _RNG_DINT;
        inst->u0 -= _RNG_DINT;
        inst->u1 -= _RNG_DINT;
        inst->u2 -= _RNG_DINT;
    }
    else if(inst->x0 < _MIN_DINT)
    {
        inst->x0 += _RNG_DINT;
        inst->x1 += _RNG_DINT;
        inst->x2 += _RNG_DINT;
        inst->u0 += _RNG_DINT;
        inst->u1 += _RNG_DINT;
        inst->u2 += _RNG_DINT;
    }

    inst->X =(signed long int)inst->x0;
    return;
}
```

#### EXT_DINT.c - Extrapolator filter
```c
/********************************************************************
 * COPYRIGHT -- Bernecker + Rainer
 ********************************************************************
 * Library: FiltLib
 * File: EXT_DINT.c
 * Author: passaglial
 * Created: August 29, 2012
 ********************************************************************
 * Implementation of library FiltLib
 ********************************************************************/

#include <bur/plctypes.h>
#include <math.h>
#ifdef __cplusplus
	extern "C"
	{
#endif

	#include "FiltLib.h"
    #include "Filtlib_defines.h"

#ifdef __cplusplus
	};
#endif

/* Auxiliary functions */
static void fnInitExtDint(struct EXT_DINT* inst);
static void fnCalcExtDint(struct EXT_DINT* inst);
static void fnCoeffExt(struct EXT_DINT* inst);

/* Extrapolator filter */
void EXT_DINT(struct EXT_DINT* inst)
{
    if(inst->Enable == 0) /* Not enabled? */
    {
        inst->Busy = 0;
        inst->Valid = 0;
        inst->Error = 0;
        inst->ErrorID = 0;
        inst->X = 0;
        return;
    }
    else if(inst->Busy == 0) /* Just enabled? */
    {
        inst->Busy = 1;
        fnInitExtDint(inst);
    }

    /*** FB is enabled ***/

    if(inst->Error != 0)
    {
        inst->Busy = 1;
        inst->Valid = 0;
        return;
    }

    fnCalcExtDint(inst);

    inst->Busy = 1;
    inst->Valid = 1;
    return;
}

static void fnInitExtDint(struct EXT_DINT* inst)
{
    RTInfo_typ rti;

    rti.enable = 1;
    RTInfo(&rti);

    if(rti.status != ERR_OK)
    {
        inst->ErrorID = FLTLIB_ER_GET_TASKTIME;
        inst->Error = 1;
        return;
    }

    inst->Ts = (double)rti.cycle_time * 1E-6;

    if(inst->T_ext < 1.5 * inst->Ts)
    {
        inst->Error = 1;
        inst->ErrorID = FLTLIB_ER_EXT_TIME_TOO_LOW;
        return;
    }

    fnCoeffExt(inst);

    inst->u0 = (double)inst->U;
    inst->u1 = inst->u0;
    inst->x0 = inst->u0;
    inst->x1 = inst->u0;
    inst->U_old = (long signed int)inst->u0;
    return;
}

static void fnCoeffExt(struct EXT_DINT* inst)
{
    /* Temporary variables */
    double k, h, alpha, Tz1, Tz2, Tp, a0, m1, m2, q1, q2, r, rr;

    /* Initizlization  */
    k = 4;

    /* Zero at highest frequency */
    Tz2 = k * inst->Ts;

    /* alpha comptation (distance between singularities) */
    h = sqrt(Tz2 / inst->T_ext);
    alpha = h / (h + 1);

    /* Poles and Zeros for continuos time Transfer function */
    Tp  = Tz2 / alpha;
    Tz1 = Tz2 / (alpha * alpha);

    /* Auxiliary parameters */
    m1 = Tz1 + Tz2;
    m2 = Tz1 * Tz2;
    q1 = 2 * Tp;
    q2 = Tp * Tp;
    r = 2 / inst->Ts;
    rr = r * r;

    /* Coefficients for discrete time transfer function */
    a0 = 1 + r*q1 + rr*q2;
    inst->a1 = (2 - 2*rr*q2) / a0;
    inst->a2 = (1 - r*q1 + rr*q2) / a0;
    inst->b0 = (1 + r*m1 + rr*m2) / a0;
    inst->b1 = (2 - 2*rr*m2) / a0;
    inst->b2 = (1 - r*m1 + rr*m2) / a0;

    return;
}

static void fnCalcExtDint(struct EXT_DINT* inst)
{

    inst->x2 = inst->x1;
    inst->x1 = inst->x0;
    inst->u2 = inst->u1;
    inst->u1 = inst->u0;
    inst->u0 += (double)(inst->U - inst->U_old);
    inst->U_old = inst->U;

    inst->x0 = -(inst->a1 * inst->x1) -(inst->a2 * inst->x2)
        +(inst->b0 * inst->u0) +(inst->b1 * inst->u1) +(inst->b2 * inst->u2);

    if(inst->x0 > _MAX_DINT)
    {
        inst->x0 -= _RNG_DINT;
        inst->x1 -= _RNG_DINT;
        inst->x2 -= _RNG_DINT;
        inst->u0 -= _RNG_DINT;
        inst->u1 -= _RNG_DINT;
        inst->u2 -= _RNG_DINT;
    }
    else if(inst->x0 < _MIN_DINT)
    {
        inst->x0 += _RNG_DINT;
        inst->x1 += _RNG_DINT;
        inst->x2 += _RNG_DINT;
        inst->u0 += _RNG_DINT;
        inst->u1 += _RNG_DINT;
        inst->u2 += _RNG_DINT;
    }

    inst->X =(signed long int)inst->x0;
    return;
}
```

#### FDT_DINT.c - Generic Transfer function
```c
/********************************************************************
 * COPYRIGHT --
 ********************************************************************
 * Library: FiltLib
 * File: FDT_DINT.c
 * Author: passaglial
 * Created: September 08, 2010
 ********************************************************************
 * Implementation of library FiltLib
 ********************************************************************/

#include <bur/plctypes.h>
#include "FiltLib.h"
#include "Filtlib_defines.h"

/* Auxiliary functions */
static void fnInitFdtDint(struct FDT_DINT* inst);
static void fnCalcFdtDint(struct FDT_DINT* inst);

/*Generic Transfer function*/
void FDT_DINT(struct FDT_DINT* inst)
{
    if(inst->Enable == 0) /* Not enabled? */
    {
        inst->Busy = 0;
        inst->Valid = 0;
        inst->Error = 0;
        inst->ErrorID = 0;
        inst->X = 0;
        return;
    }
    else if(inst->Busy == 0) /* Just enabled? */
    {
       inst->Busy = 1;
       fnInitFdtDint(inst);
    }

    /*** FB is enabled ***/

    if(inst->Error != 0)
    {
        inst->Busy = 1;
        inst->Valid = 0;
        return;
    }

    fnCalcFdtDint(inst);

    inst->Busy = 1;
    inst->Valid = 1;
    return;

}

static void fnInitFdtDint(struct FDT_DINT* inst)
{
    inst->u0 = (double)inst->U;
    inst->u1 = inst->u0;
    inst->x0 = inst->u0;
    inst->x1 = inst->u0;
    inst->U_old = (long signed int)inst->u0;
    return;
}

static void fnCalcFdtDint(struct FDT_DINT* inst)
{

    inst->x2 = inst->x1;
    inst->x1 = inst->x0;
    inst->u2 = inst->u1;
    inst->u1 = inst->u0;
    inst->u0 += (double)(inst->U - inst->U_old);
    inst->U_old = inst->U;

    inst->x0 = -(inst->a1 * inst->x1) -(inst->a2 * inst->x2)
               +(inst->b0 * inst->u0) +(inst->b1 * inst->u1) +(inst->b2 * inst->u2);

    if(inst->x0 > _MAX_DINT)
    {
        inst->x0 -= _RNG_DINT;
        inst->x1 -= _RNG_DINT;
        inst->x2 -= _RNG_DINT;
        inst->u0 -= _RNG_DINT;
        inst->u1 -= _RNG_DINT;
        inst->u2 -= _RNG_DINT;
    }
    else if(inst->x0 < _MIN_DINT)
    {
        inst->x0 += _RNG_DINT;
        inst->x1 += _RNG_DINT;
        inst->x2 += _RNG_DINT;
        inst->u0 += _RNG_DINT;
        inst->u1 += _RNG_DINT;
        inst->u2 += _RNG_DINT;
    }

    inst->X =(signed long int)inst->x0;
    return;
}
```

### Package Logical/30_MC/Task - Tasks

### Package Logical/30_MC/Task/Cyclic01 - Package

### Program Logical/30_MC/Task/Cyclic01/MC_HIERARCHY (IEC) - MC_HIERARCHY - C#1 (0.8ms)
